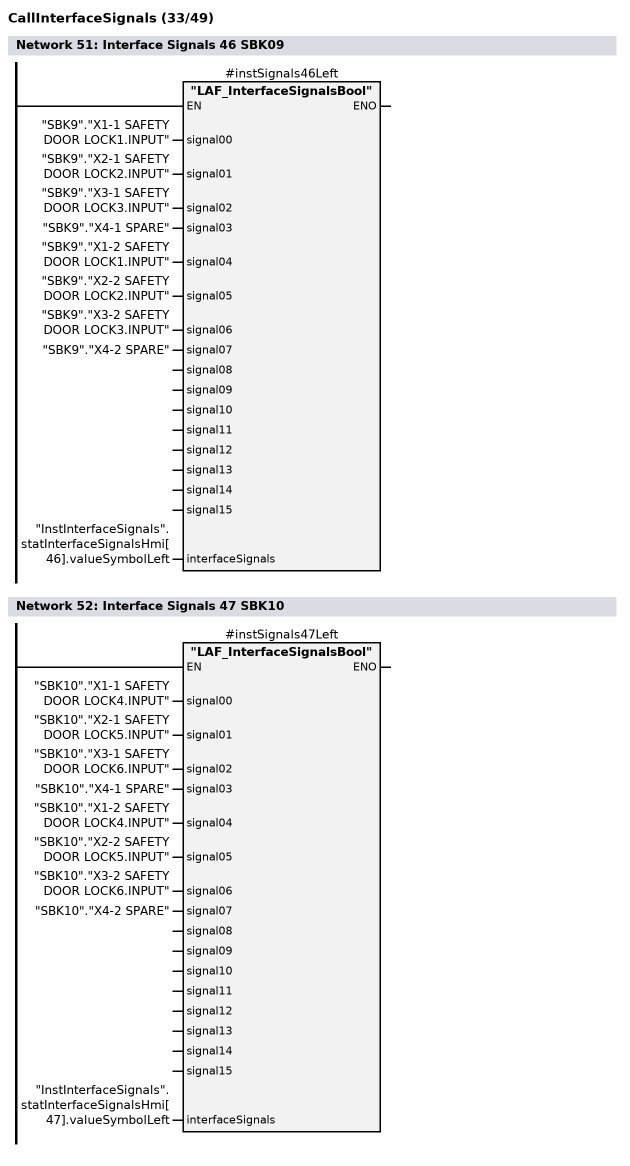
   RUNG wire#powerrail
      #instSignals46Left(signal00 := "SBK9"."X1-1 SAFETY DOOR LOCK1.INPUT", signal01 := "SBK9"."X2-1 SAFETY DOOR LOCK2.INPUT", signal02 := "SBK9"."X3-1 SAFETY DOOR LOCK3.INPUT", signal03 := "SBK9"."X4-1 SPARE", signal04 := "SBK9"."X1-2 SAFETY DOOR LOCK1.INPUT", signal05 := "SBK9"."X2-2 SAFETY DOOR LOCK2.INPUT", signal06 := "SBK9"."X3-2 SAFETY DOOR LOCK3.INPUT", signal07 := "SBK9"."X4-2 SPARE", signal08 :=, signal09 :=, signal10 :=, signal11 :=, signal12 :=, signal13 :=, signal14 :=, signal15 :=, interfaceSignals := "InstInterfaceSignals".statInterfaceSignalsHmi[46].valueSymbolLeft)
   END_RUNG
   // the same network as SCL:
   #instSignals46Left(signal00 := "SBK9"."X1-1 SAFETY DOOR LOCK1.INPUT",   // "LAF_InterfaceSignalsBool"
                      signal01 := "SBK9"."X2-1 SAFETY DOOR LOCK2.INPUT",
                      signal02 := "SBK9"."X3-1 SAFETY DOOR LOCK3.INPUT",
                      signal03 := "SBK9"."X4-1 SPARE",
                      signal04 := "SBK9"."X1-2 SAFETY DOOR LOCK1.INPUT",
                      signal05 := "SBK9"."X2-2 SAFETY DOOR LOCK2.INPUT",
                      signal06 := "SBK9"."X3-2 SAFETY DOOR LOCK3.INPUT",
                      signal07 := "SBK9"."X4-2 SPARE",
                      interfaceSignals := "InstInterfaceSignals".statInterfaceSignalsHmi[46].valueSymbolLeft);
END_REGION

REGION Network 52: Interface Signals 47 SBK10
   RUNG wire#powerrail
      #instSignals47Left(signal00 := "SBK10"."X1-1 SAFETY DOOR LOCK4.INPUT", signal01 := "SBK10"."X2-1 SAFETY DOOR LOCK5.INPUT", signal02 := "SBK10"."X3-1 SAFETY DOOR LOCK6.INPUT", signal03 := "SBK10"."X4-1 SPARE", signal04 := "SBK10"."X1-2 SAFETY DOOR LOCK4.INPUT", signal05 := "SBK10"."X2-2 SAFETY DOOR LOCK5.INPUT", signal06 := "SBK10"."X3-2 SAFETY DOOR LOCK6.INPUT", signal07 := "SBK10"."X4-2 SPARE", signal08 :=, signal09 :=, signal10 :=, signal11 :=, signal12 :=, signal13 :=, signal14 :=, signal15 :=, interfaceSignals := "InstInterfaceSignals".statInterfaceSignalsHmi[47].valueSymbolLeft)
   END_RUNG
   // the same network as SCL:
   #instSignals47Left(signal00 := "SBK10"."X1-1 SAFETY DOOR LOCK4.INPUT",   // "LAF_InterfaceSignalsBool"
                      signal01 := "SBK10"."X2-1 SAFETY DOOR LOCK5.INPUT",
                      signal02 := "SBK10"."X3-1 SAFETY DOOR LOCK6.INPUT",
                      signal03 := "SBK10"."X4-1 SPARE",
                      signal04 := "SBK10"."X1-2 SAFETY DOOR LOCK4.INPUT",
                      signal05 := "SBK10"."X2-2 SAFETY DOOR LOCK5.INPUT",
                      signal06 := "SBK10"."X3-2 SAFETY DOOR LOCK6.INPUT",
                      signal07 := "SBK10"."X4-2 SPARE",
                      interfaceSignals := "InstInterfaceSignals".statInterfaceSignalsHmi[47].valueSymbolLeft);
END_REGION

REGION Network 53: Interface Signals 48 SBK11
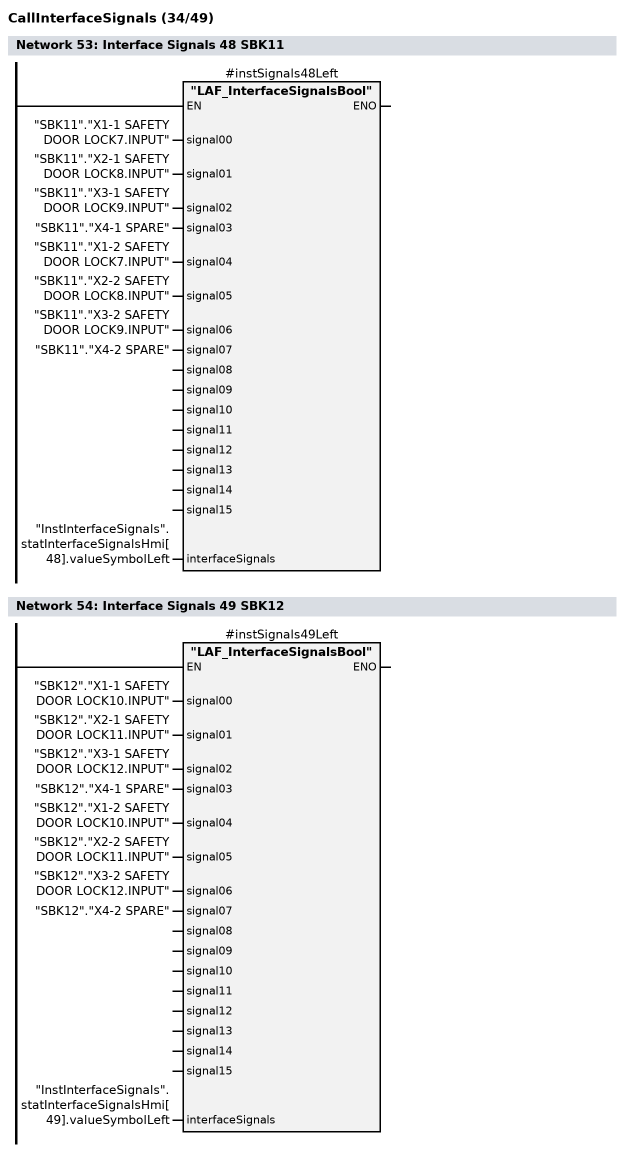
   RUNG wire#powerrail
      #instSignals48Left(signal00 := "SBK11"."X1-1 SAFETY DOOR LOCK7.INPUT", signal01 := "SBK11"."X2-1 SAFETY DOOR LOCK8.INPUT", signal02 := "SBK11"."X3-1 SAFETY DOOR LOCK9.INPUT", signal03 := "SBK11"."X4-1 SPARE", signal04 := "SBK11"."X1-2 SAFETY DOOR LOCK7.INPUT", signal05 := "SBK11"."X2-2 SAFETY DOOR LOCK8.INPUT", signal06 := "SBK11"."X3-2 SAFETY DOOR LOCK9.INPUT", signal07 := "SBK11"."X4-2 SPARE", signal08 :=, signal09 :=, signal10 :=, signal11 :=, signal12 :=, signal13 :=, signal14 :=, signal15 :=, interfaceSignals := "InstInterfaceSignals".statInterfaceSignalsHmi[48].valueSymbolLeft)
   END_RUNG
   // the same network as SCL:
   #instSignals48Left(signal00 := "SBK11"."X1-1 SAFETY DOOR LOCK7.INPUT",   // "LAF_InterfaceSignalsBool"
                      signal01 := "SBK11"."X2-1 SAFETY DOOR LOCK8.INPUT",
                      signal02 := "SBK11"."X3-1 SAFETY DOOR LOCK9.INPUT",
                      signal03 := "SBK11"."X4-1 SPARE",
                      signal04 := "SBK11"."X1-2 SAFETY DOOR LOCK7.INPUT",
                      signal05 := "SBK11"."X2-2 SAFETY DOOR LOCK8.INPUT",
                      signal06 := "SBK11"."X3-2 SAFETY DOOR LOCK9.INPUT",
                      signal07 := "SBK11"."X4-2 SPARE",
                      interfaceSignals := "InstInterfaceSignals".statInterfaceSignalsHmi[48].valueSymbolLeft);
END_REGION

REGION Network 54: Interface Signals 49 SBK12
   RUNG wire#powerrail
      #instSignals49Left(signal00 := "SBK12"."X1-1 SAFETY DOOR LOCK10.INPUT", signal01 := "SBK12"."X2-1 SAFETY DOOR LOCK11.INPUT", signal02 := "SBK12"."X3-1 SAFETY DOOR LOCK12.INPUT", signal03 := "SBK12"."X4-1 SPARE", signal04 := "SBK12"."X1-2 SAFETY DOOR LOCK10.INPUT", signal05 := "SBK12"."X2-2 SAFETY DOOR LOCK11.INPUT", signal06 := "SBK12"."X3-2 SAFETY DOOR LOCK12.INPUT", signal07 := "SBK12"."X4-2 SPARE", signal08 :=, signal09 :=, signal10 :=, signal11 :=, signal12 :=, signal13 :=, signal14 :=, signal15 :=, interfaceSignals := "InstInterfaceSignals".statInterfaceSignalsHmi[49].valueSymbolLeft)
   END_RUNG
   // the same network as SCL:
   #instSignals49Left(signal00 := "SBK12"."X1-1 SAFETY DOOR LOCK10.INPUT",   // "LAF_InterfaceSignalsBool"
                      signal01 := "SBK12"."X2-1 SAFETY DOOR LOCK11.INPUT",
                      signal02 := "SBK12"."X3-1 SAFETY DOOR LOCK12.INPUT",
                      signal03 := "SBK12"."X4-1 SPARE",
                      signal04 := "SBK12"."X1-2 SAFETY DOOR LOCK10.INPUT",
                      signal05 := "SBK12"."X2-2 SAFETY DOOR LOCK11.INPUT",
                      signal06 := "SBK12"."X3-2 SAFETY DOOR LOCK12.INPUT",
                      signal07 := "SBK12"."X4-2 SPARE",
                      interfaceSignals := "InstInterfaceSignals".statInterfaceSignalsHmi[49].valueSymbolLeft);
END_REGION

REGION Network 55: Interface Signals 50 SBK13
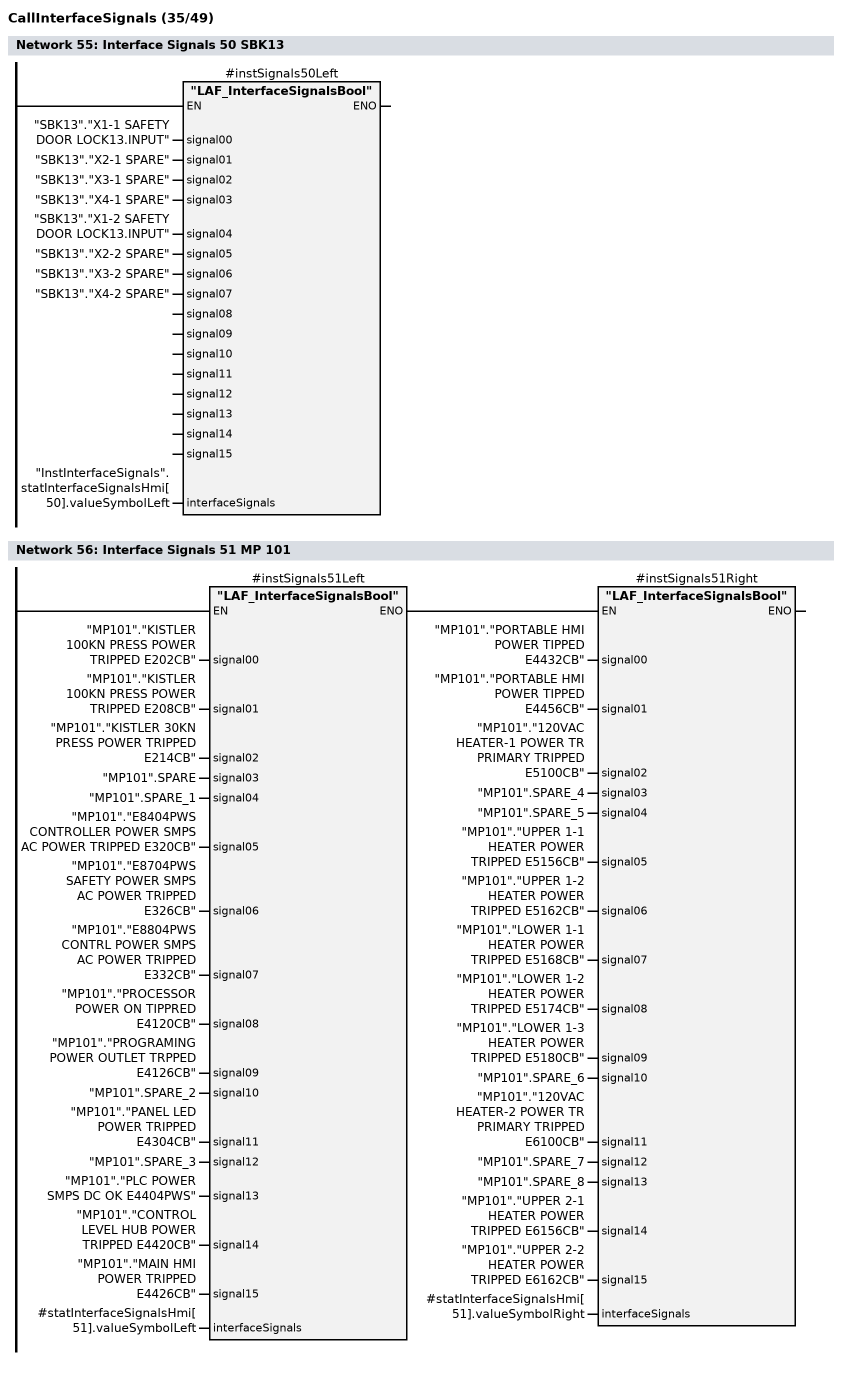
   RUNG wire#powerrail
      #instSignals50Left(signal00 := "SBK13"."X1-1 SAFETY DOOR LOCK13.INPUT", signal01 := "SBK13"."X2-1 SPARE", signal02 := "SBK13"."X3-1 SPARE", signal03 := "SBK13"."X4-1 SPARE", signal04 := "SBK13"."X1-2 SAFETY DOOR LOCK13.INPUT", signal05 := "SBK13"."X2-2 SPARE", signal06 := "SBK13"."X3-2 SPARE", signal07 := "SBK13"."X4-2 SPARE", signal08 :=, signal09 :=, signal10 :=, signal11 :=, signal12 :=, signal13 :=, signal14 :=, signal15 :=, interfaceSignals := "InstInterfaceSignals".statInterfaceSignalsHmi[50].valueSymbolLeft)
   END_RUNG
   // the same network as SCL:
   #instSignals50Left(signal00 := "SBK13"."X1-1 SAFETY DOOR LOCK13.INPUT",   // "LAF_InterfaceSignalsBool"
                      signal01 := "SBK13"."X2-1 SPARE",
                      signal02 := "SBK13"."X3-1 SPARE",
                      signal03 := "SBK13"."X4-1 SPARE",
                      signal04 := "SBK13"."X1-2 SAFETY DOOR LOCK13.INPUT",
                      signal05 := "SBK13"."X2-2 SPARE",
                      signal06 := "SBK13"."X3-2 SPARE",
                      signal07 := "SBK13"."X4-2 SPARE",
                      interfaceSignals := "InstInterfaceSignals".statInterfaceSignalsHmi[50].valueSymbolLeft);
END_REGION

REGION Network 56: Interface Signals 51 MP 101
   RUNG wire#powerrail
      #instSignals51Left(signal00 := "MP101"."KISTLER 100KN PRESS POWER TRIPPED E202CB", signal01 := "MP101"."KISTLER 100KN PRESS POWER TRIPPED E208CB", signal02 := "MP101"."KISTLER 30KN PRESS POWER TRIPPED E214CB", signal03 := "MP101".SPARE, signal04 := "MP101".SPARE_1, signal05 := "MP101"."E8404PWS CONTROLLER POWER SMPS AC POWER TRIPPED E320CB", signal06 := "MP101"."E8704PWS SAFETY POWER SMPS AC POWER TRIPPED E326CB", signal07 := "MP101"."E8804PWS CONTRL POWER SMPS AC POWER TRIPPED E332CB", signal08 := "MP101"."PROCESSOR POWER ON TIPPRED E4120CB", signal09 := "MP101"."PROGRAMING POWER OUTLET TRPPED E4126CB", signal10 := "MP101".SPARE_2, signal11 := "MP101"."PANEL LED POWER TRIPPED E4304CB", signal12 := "MP101".SPARE_3, signal13 := "MP101"."PLC POWER SMPS DC OK E4404PWS", signal14 := "MP101"."CONTROL LEVEL HUB POWER TRIPPED E4420CB", signal15 := "MP101"."MAIN HMI POWER TRIPPED E4426CB", interfaceSignals := #statInterfaceSignalsHmi[51].valueSymbolLeft)
      #instSignals51Right(signal00 := "MP101"."PORTABLE HMI POWER TIPPED E4432CB", signal01 := "MP101"."PORTABLE HMI POWER TIPPED E4456CB", signal02 := "MP101"."120VAC HEATER-1 POWER TR PRIMARY TRIPPED E5100CB", signal03 := "MP101".SPARE_4, signal04 := "MP101".SPARE_5, signal05 := "MP101"."UPPER 1-1 HEATER POWER TRIPPED E5156CB", signal06 := "MP101"."UPPER 1-2 HEATER POWER TRIPPED E5162CB", signal07 := "MP101"."LOWER 1-1 HEATER POWER TRIPPED E5168CB", signal08 := "MP101"."LOWER 1-2 HEATER POWER TRIPPED E5174CB", signal09 := "MP101"."LOWER 1-3 HEATER POWER TRIPPED E5180CB", signal10 := "MP101".SPARE_6, signal11 := "MP101"."120VAC HEATER-2 POWER TR PRIMARY TRIPPED E6100CB", signal12 := "MP101".SPARE_7, signal13 := "MP101".SPARE_8, signal14 := "MP101"."UPPER 2-1 HEATER POWER TRIPPED E6156CB", signal15 := "MP101"."UPPER 2-2 HEATER POWER TRIPPED E6162CB", interfaceSignals := #statInterfaceSignalsHmi[51].valueSymbolRight)
   END_RUNG
   // the same network as SCL:
   #instSignals51Left(signal00 := "MP101"."KISTLER 100KN PRESS POWER TRIPPED E202CB",   // "LAF_InterfaceSignalsBool"
                      signal01 := "MP101"."KISTLER 100KN PRESS POWER TRIPPED E208CB",
                      signal02 := "MP101"."KISTLER 30KN PRESS POWER TRIPPED E214CB",
                      signal03 := "MP101".SPARE,
                      signal04 := "MP101".SPARE_1,
                      signal05 := "MP101"."E8404PWS CONTROLLER POWER SMPS AC POWER TRIPPED E320CB",
                      signal06 := "MP101"."E8704PWS SAFETY POWER SMPS AC POWER TRIPPED E326CB",
                      signal07 := "MP101"."E8804PWS CONTRL POWER SMPS AC POWER TRIPPED E332CB",
                      signal08 := "MP101"."PROCESSOR POWER ON TIPPRED E4120CB",
                      signal09 := "MP101"."PROGRAMING POWER OUTLET TRPPED E4126CB",
                      signal10 := "MP101".SPARE_2,
                      signal11 := "MP101"."PANEL LED POWER TRIPPED E4304CB",
                      signal12 := "MP101".SPARE_3,
                      signal13 := "MP101"."PLC POWER SMPS DC OK E4404PWS",
                      signal14 := "MP101"."CONTROL LEVEL HUB POWER TRIPPED E4420CB",
                      signal15 := "MP101"."MAIN HMI POWER TRIPPED E4426CB",
                      interfaceSignals := #statInterfaceSignalsHmi[51].valueSymbolLeft,
                      ENO => #_w1);
   IF #_w1 THEN
       #instSignals51Right(signal00 := "MP101"."PORTABLE HMI POWER TIPPED E4432CB",   // "LAF_InterfaceSignalsBool"
                           signal01 := "MP101"."PORTABLE HMI POWER TIPPED E4456CB",
                           signal02 := "MP101"."120VAC HEATER-1 POWER TR PRIMARY TRIPPED E5100CB",
                           signal03 := "MP101".SPARE_4,
                           signal04 := "MP101".SPARE_5,
                           signal05 := "MP101"."UPPER 1-1 HEATER POWER TRIPPED E5156CB",
                           signal06 := "MP101"."UPPER 1-2 HEATER POWER TRIPPED E5162CB",
                           signal07 := "MP101"."LOWER 1-1 HEATER POWER TRIPPED E5168CB",
                           signal08 := "MP101"."LOWER 1-2 HEATER POWER TRIPPED E5174CB",
                           signal09 := "MP101"."LOWER 1-3 HEATER POWER TRIPPED E5180CB",
                           signal10 := "MP101".SPARE_6,
                           signal11 := "MP101"."120VAC HEATER-2 POWER TR PRIMARY TRIPPED E6100CB",
                           signal12 := "MP101".SPARE_7,
                           signal13 := "MP101".SPARE_8,
                           signal14 := "MP101"."UPPER 2-1 HEATER POWER TRIPPED E6156CB",
                           signal15 := "MP101"."UPPER 2-2 HEATER POWER TRIPPED E6162CB",
                           interfaceSignals := #statInterfaceSignalsHmi[51].valueSymbolRight);
   END_IF;
END_REGION

REGION Network 57: Interface Signals 52 MP 102
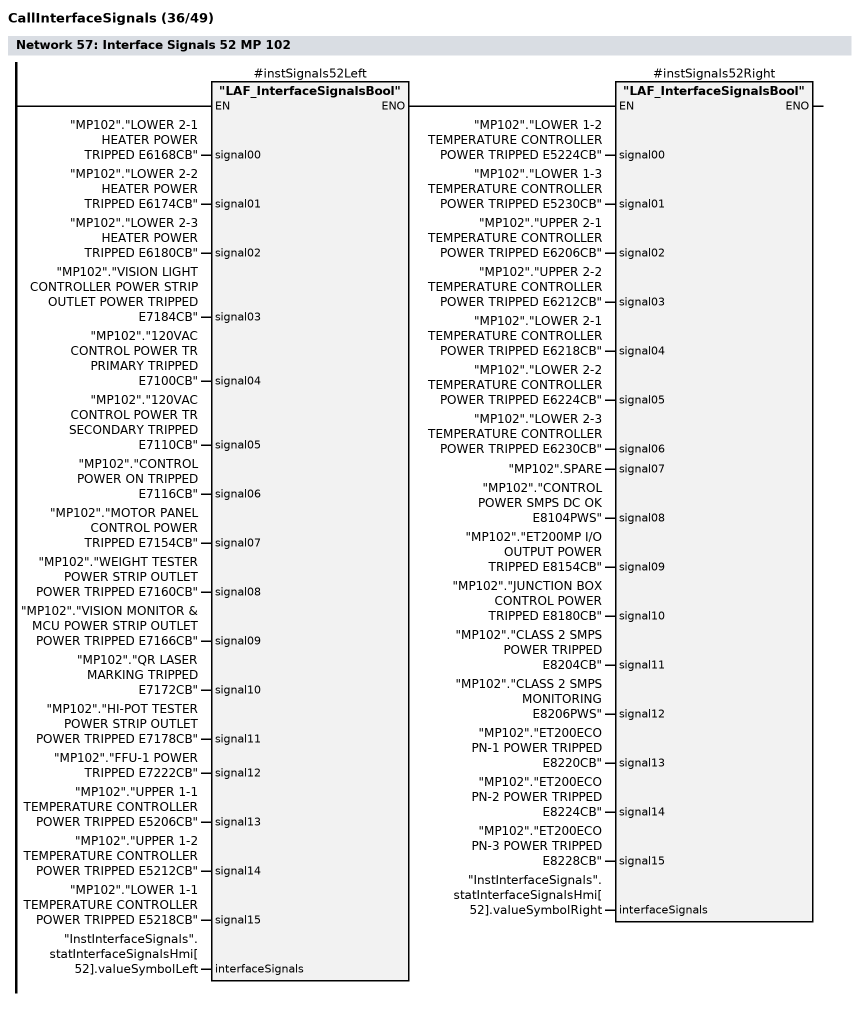
   RUNG wire#powerrail
      #instSignals52Left(signal00 := "MP102"."LOWER 2-1 HEATER POWER TRIPPED E6168CB", signal01 := "MP102"."LOWER 2-2 HEATER POWER TRIPPED E6174CB", signal02 := "MP102"."LOWER 2-3 HEATER POWER TRIPPED E6180CB", signal03 := "MP102"."VISION LIGHT CONTROLLER POWER STRIP OUTLET POWER TRIPPED E7184CB", signal04 := "MP102"."120VAC CONTROL POWER TR PRIMARY TRIPPED E7100CB", signal05 := "MP102"."120VAC CONTROL POWER TR SECONDARY TRIPPED E7110CB", signal06 := "MP102"."CONTROL POWER ON TRIPPED E7116CB", signal07 := "MP102"."MOTOR PANEL CONTROL POWER TRIPPED E7154CB", signal08 := "MP102"."WEIGHT TESTER POWER STRIP OUTLET POWER TRIPPED E7160CB", signal09 := "MP102"."VISION MONITOR & MCU POWER STRIP OUTLET POWER TRIPPED E7166CB", signal10 := "MP102"."QR LASER MARKING TRIPPED E7172CB", signal11 := "MP102"."HI-POT TESTER POWER STRIP OUTLET POWER TRIPPED E7178CB", signal12 := "MP102"."FFU-1 POWER TRIPPED E7222CB", signal13 := "MP102"."UPPER 1-1 TEMPERATURE CONTROLLER POWER TRIPPED E5206CB", signal14 := "MP102"."UPPER 1-2 TEMPERATURE CONTROLLER POWER TRIPPED E5212CB", signal15 := "MP102"."LOWER 1-1 TEMPERATURE CONTROLLER POWER TRIPPED E5218CB", interfaceSignals := "InstInterfaceSignals".statInterfaceSignalsHmi[52].valueSymbolLeft)
      #instSignals52Right(signal00 := "MP102"."LOWER 1-2 TEMPERATURE CONTROLLER POWER TRIPPED E5224CB", signal01 := "MP102"."LOWER 1-3 TEMPERATURE CONTROLLER POWER TRIPPED E5230CB", signal02 := "MP102"."UPPER 2-1 TEMPERATURE CONTROLLER POWER TRIPPED E6206CB", signal03 := "MP102"."UPPER 2-2 TEMPERATURE CONTROLLER POWER TRIPPED E6212CB", signal04 := "MP102"."LOWER 2-1 TEMPERATURE CONTROLLER POWER TRIPPED E6218CB", signal05 := "MP102"."LOWER 2-2 TEMPERATURE CONTROLLER POWER TRIPPED E6224CB", signal06 := "MP102"."LOWER 2-3 TEMPERATURE CONTROLLER POWER TRIPPED E6230CB", signal07 := "MP102".SPARE, signal08 := "MP102"."CONTROL POWER SMPS DC OK E8104PWS", signal09 := "MP102"."ET200MP I/O OUTPUT POWER TRIPPED E8154CB", signal10 := "MP102"."JUNCTION BOX CONTROL POWER TRIPPED E8180CB", signal11 := "MP102"."CLASS 2 SMPS POWER TRIPPED E8204CB", signal12 := "MP102"."CLASS 2 SMPS MONITORING E8206PWS", signal13 := "MP102"."ET200ECO PN-1 POWER TRIPPED E8220CB", signal14 := "MP102"."ET200ECO PN-2 POWER TRIPPED E8224CB", signal15 := "MP102"."ET200ECO PN-3 POWER TRIPPED E8228CB", interfaceSignals := "InstInterfaceSignals".statInterfaceSignalsHmi[52].valueSymbolRight)
   END_RUNG
   // the same network as SCL:
   #instSignals52Left(signal00 := "MP102"."LOWER 2-1 HEATER POWER TRIPPED E6168CB",   // "LAF_InterfaceSignalsBool"
                      signal01 := "MP102"."LOWER 2-2 HEATER POWER TRIPPED E6174CB",
                      signal02 := "MP102"."LOWER 2-3 HEATER POWER TRIPPED E6180CB",
                      signal03 := "MP102"."VISION LIGHT CONTROLLER POWER STRIP OUTLET POWER TRIPPED E7184CB",
                      signal04 := "MP102"."120VAC CONTROL POWER TR PRIMARY TRIPPED E7100CB",
                      signal05 := "MP102"."120VAC CONTROL POWER TR SECONDARY TRIPPED E7110CB",
                      signal06 := "MP102"."CONTROL POWER ON TRIPPED E7116CB",
                      signal07 := "MP102"."MOTOR PANEL CONTROL POWER TRIPPED E7154CB",
                      signal08 := "MP102"."WEIGHT TESTER POWER STRIP OUTLET POWER TRIPPED E7160CB",
                      signal09 := "MP102"."VISION MONITOR & MCU POWER STRIP OUTLET POWER TRIPPED E7166CB",
                      signal10 := "MP102"."QR LASER MARKING TRIPPED E7172CB",
                      signal11 := "MP102"."HI-POT TESTER POWER STRIP OUTLET POWER TRIPPED E7178CB",
                      signal12 := "MP102"."FFU-1 POWER TRIPPED E7222CB",
                      signal13 := "MP102"."UPPER 1-1 TEMPERATURE CONTROLLER POWER TRIPPED E5206CB",
                      signal14 := "MP102"."UPPER 1-2 TEMPERATURE CONTROLLER POWER TRIPPED E5212CB",
                      signal15 := "MP102"."LOWER 1-1 TEMPERATURE CONTROLLER POWER TRIPPED E5218CB",
                      interfaceSignals := "InstInterfaceSignals".statInterfaceSignalsHmi[52].valueSymbolLeft,
                      ENO => #_w1);
   IF #_w1 THEN
       #instSignals52Right(signal00 := "MP102"."LOWER 1-2 TEMPERATURE CONTROLLER POWER TRIPPED E5224CB",   // "LAF_InterfaceSignalsBool"
                           signal01 := "MP102"."LOWER 1-3 TEMPERATURE CONTROLLER POWER TRIPPED E5230CB",
                           signal02 := "MP102"."UPPER 2-1 TEMPERATURE CONTROLLER POWER TRIPPED E6206CB",
                           signal03 := "MP102"."UPPER 2-2 TEMPERATURE CONTROLLER POWER TRIPPED E6212CB",
                           signal04 := "MP102"."LOWER 2-1 TEMPERATURE CONTROLLER POWER TRIPPED E6218CB",
                           signal05 := "MP102"."LOWER 2-2 TEMPERATURE CONTROLLER POWER TRIPPED E6224CB",
                           signal06 := "MP102"."LOWER 2-3 TEMPERATURE CONTROLLER POWER TRIPPED E6230CB",
                           signal07 := "MP102".SPARE,
                           signal08 := "MP102"."CONTROL POWER SMPS DC OK E8104PWS",
                           signal09 := "MP102"."ET200MP I/O OUTPUT POWER TRIPPED E8154CB",
                           signal10 := "MP102"."JUNCTION BOX CONTROL POWER TRIPPED E8180CB",
                           signal11 := "MP102"."CLASS 2 SMPS POWER TRIPPED E8204CB",
                           signal12 := "MP102"."CLASS 2 SMPS MONITORING E8206PWS",
                           signal13 := "MP102"."ET200ECO PN-1 POWER TRIPPED E8220CB",
                           signal14 := "MP102"."ET200ECO PN-2 POWER TRIPPED E8224CB",
                           signal15 := "MP102"."ET200ECO PN-3 POWER TRIPPED E8228CB",
                           interfaceSignals := "InstInterfaceSignals".statInterfaceSignalsHmi[52].valueSymbolRight);
   END_IF;
END_REGION

REGION Network 58: Interface Signals 53 MP 103
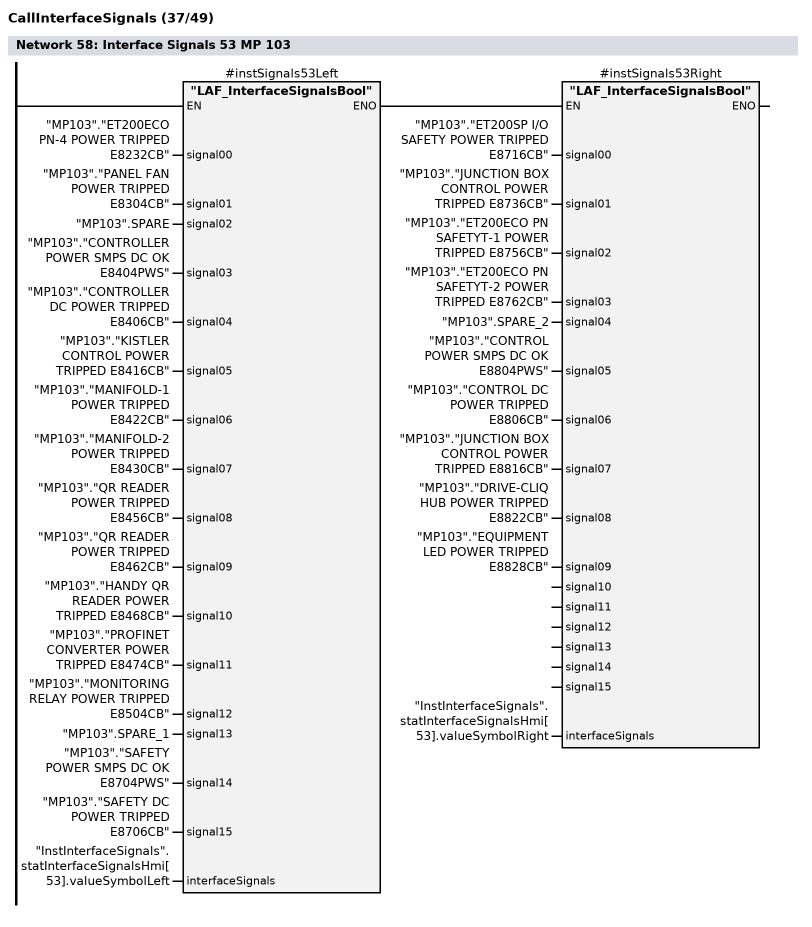
   RUNG wire#powerrail
      #instSignals53Left(signal00 := "MP103"."ET200ECO PN-4 POWER TRIPPED E8232CB", signal01 := "MP103"."PANEL FAN POWER TRIPPED E8304CB", signal02 := "MP103".SPARE, signal03 := "MP103"."CONTROLLER POWER SMPS DC OK E8404PWS", signal04 := "MP103"."CONTROLLER DC POWER TRIPPED E8406CB", signal05 := "MP103"."KISTLER CONTROL POWER TRIPPED E8416CB", signal06 := "MP103"."MANIFOLD-1 POWER TRIPPED E8422CB", signal07 := "MP103"."MANIFOLD-2 POWER TRIPPED E8430CB", signal08 := "MP103"."QR READER POWER TRIPPED E8456CB", signal09 := "MP103"."QR READER POWER TRIPPED E8462CB", signal10 := "MP103"."HANDY QR READER POWER TRIPPED E8468CB", signal11 := "MP103"."PROFINET CONVERTER POWER TRIPPED E8474CB", signal12 := "MP103"."MONITORING RELAY POWER TRIPPED E8504CB", signal13 := "MP103".SPARE_1, signal14 := "MP103"."SAFETY POWER SMPS DC OK E8704PWS", signal15 := "MP103"."SAFETY DC POWER TRIPPED E8706CB", interfaceSignals := "InstInterfaceSignals".statInterfaceSignalsHmi[53].valueSymbolLeft)
      #instSignals53Right(signal00 := "MP103"."ET200SP I/O SAFETY POWER TRIPPED E8716CB", signal01 := "MP103"."JUNCTION BOX CONTROL POWER TRIPPED E8736CB", signal02 := "MP103"."ET200ECO PN SAFETYT-1 POWER TRIPPED E8756CB", signal03 := "MP103"."ET200ECO PN SAFETYT-2 POWER TRIPPED E8762CB", signal04 := "MP103".SPARE_2, signal05 := "MP103"."CONTROL POWER SMPS DC OK E8804PWS", signal06 := "MP103"."CONTROL DC POWER TRIPPED E8806CB", signal07 := "MP103"."JUNCTION BOX CONTROL POWER TRIPPED E8816CB", signal08 := "MP103"."DRIVE-CLIQ HUB POWER TRIPPED E8822CB", signal09 := "MP103"."EQUIPMENT LED POWER TRIPPED E8828CB", signal10 :=, signal11 :=, signal12 :=, signal13 :=, signal14 :=, signal15 :=, interfaceSignals := "InstInterfaceSignals".statInterfaceSignalsHmi[53].valueSymbolRight)
   END_RUNG
   // the same network as SCL:
   #instSignals53Left(signal00 := "MP103"."ET200ECO PN-4 POWER TRIPPED E8232CB",   // "LAF_InterfaceSignalsBool"
                      signal01 := "MP103"."PANEL FAN POWER TRIPPED E8304CB",
                      signal02 := "MP103".SPARE,
                      signal03 := "MP103"."CONTROLLER POWER SMPS DC OK E8404PWS",
                      signal04 := "MP103"."CONTROLLER DC POWER TRIPPED E8406CB",
                      signal05 := "MP103"."KISTLER CONTROL POWER TRIPPED E8416CB",
                      signal06 := "MP103"."MANIFOLD-1 POWER TRIPPED E8422CB",
                      signal07 := "MP103"."MANIFOLD-2 POWER TRIPPED E8430CB",
                      signal08 := "MP103"."QR READER POWER TRIPPED E8456CB",
                      signal09 := "MP103"."QR READER POWER TRIPPED E8462CB",
                      signal10 := "MP103"."HANDY QR READER POWER TRIPPED E8468CB",
                      signal11 := "MP103"."PROFINET CONVERTER POWER TRIPPED E8474CB",
                      signal12 := "MP103"."MONITORING RELAY POWER TRIPPED E8504CB",
                      signal13 := "MP103".SPARE_1,
                      signal14 := "MP103"."SAFETY POWER SMPS DC OK E8704PWS",
                      signal15 := "MP103"."SAFETY DC POWER TRIPPED E8706CB",
                      interfaceSignals := "InstInterfaceSignals".statInterfaceSignalsHmi[53].valueSymbolLeft,
                      ENO => #_w1);
   IF #_w1 THEN
       #instSignals53Right(signal00 := "MP103"."ET200SP I/O SAFETY POWER TRIPPED E8716CB",   // "LAF_InterfaceSignalsBool"
                           signal01 := "MP103"."JUNCTION BOX CONTROL POWER TRIPPED E8736CB",
                           signal02 := "MP103"."ET200ECO PN SAFETYT-1 POWER TRIPPED E8756CB",
                           signal03 := "MP103"."ET200ECO PN SAFETYT-2 POWER TRIPPED E8762CB",
                           signal04 := "MP103".SPARE_2,
                           signal05 := "MP103"."CONTROL POWER SMPS DC OK E8804PWS",
                           signal06 := "MP103"."CONTROL DC POWER TRIPPED E8806CB",
                           signal07 := "MP103"."JUNCTION BOX CONTROL POWER TRIPPED E8816CB",
                           signal08 := "MP103"."DRIVE-CLIQ HUB POWER TRIPPED E8822CB",
                           signal09 := "MP103"."EQUIPMENT LED POWER TRIPPED E8828CB",
                           interfaceSignals := "InstInterfaceSignals".statInterfaceSignalsHmi[53].valueSymbolRight);
   END_IF;
END_REGION

REGION Network 59: Interface Signals 54 MP 104
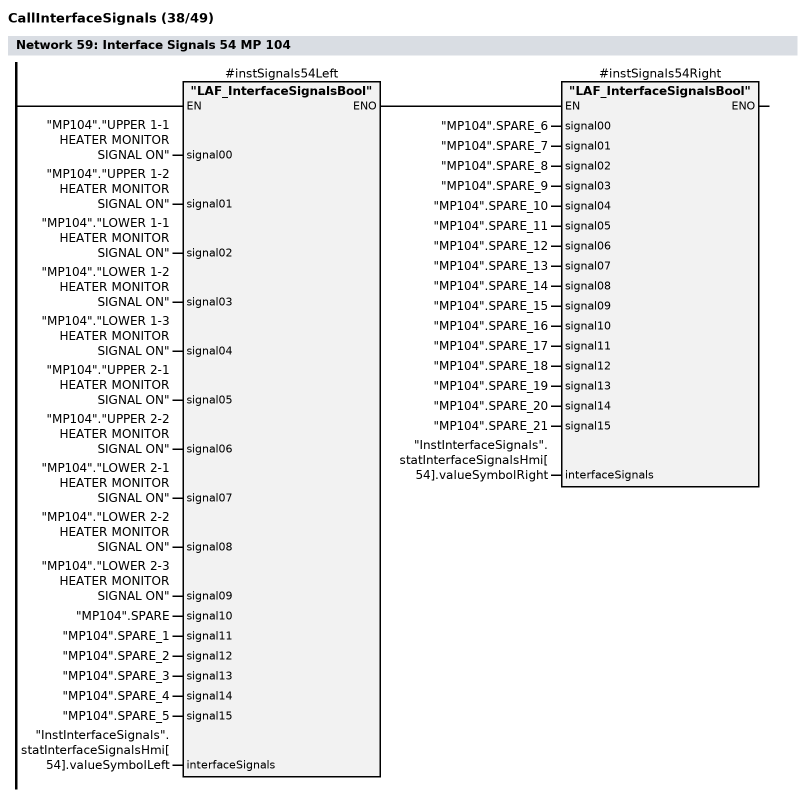
   RUNG wire#powerrail
      #instSignals54Left(signal00 := "MP104"."UPPER 1-1 HEATER MONITOR SIGNAL ON", signal01 := "MP104"."UPPER 1-2 HEATER MONITOR SIGNAL ON", signal02 := "MP104"."LOWER 1-1 HEATER MONITOR SIGNAL ON", signal03 := "MP104"."LOWER 1-2 HEATER MONITOR SIGNAL ON", signal04 := "MP104"."LOWER 1-3 HEATER MONITOR SIGNAL ON", signal05 := "MP104"."UPPER 2-1 HEATER MONITOR SIGNAL ON", signal06 := "MP104"."UPPER 2-2 HEATER MONITOR SIGNAL ON", signal07 := "MP104"."LOWER 2-1 HEATER MONITOR SIGNAL ON", signal08 := "MP104"."LOWER 2-2 HEATER MONITOR SIGNAL ON", signal09 := "MP104"."LOWER 2-3 HEATER MONITOR SIGNAL ON", signal10 := "MP104".SPARE, signal11 := "MP104".SPARE_1, signal12 := "MP104".SPARE_2, signal13 := "MP104".SPARE_3, signal14 := "MP104".SPARE_4, signal15 := "MP104".SPARE_5, interfaceSignals := "InstInterfaceSignals".statInterfaceSignalsHmi[54].valueSymbolLeft)
      #instSignals54Right(signal00 := "MP104".SPARE_6, signal01 := "MP104".SPARE_7, signal02 := "MP104".SPARE_8, signal03 := "MP104".SPARE_9, signal04 := "MP104".SPARE_10, signal05 := "MP104".SPARE_11, signal06 := "MP104".SPARE_12, signal07 := "MP104".SPARE_13, signal08 := "MP104".SPARE_14, signal09 := "MP104".SPARE_15, signal10 := "MP104".SPARE_16, signal11 := "MP104".SPARE_17, signal12 := "MP104".SPARE_18, signal13 := "MP104".SPARE_19, signal14 := "MP104".SPARE_20, signal15 := "MP104".SPARE_21, interfaceSignals := "InstInterfaceSignals".statInterfaceSignalsHmi[54].valueSymbolRight)
   END_RUNG
   // the same network as SCL:
   #instSignals54Left(signal00 := "MP104"."UPPER 1-1 HEATER MONITOR SIGNAL ON",   // "LAF_InterfaceSignalsBool"
                      signal01 := "MP104"."UPPER 1-2 HEATER MONITOR SIGNAL ON",
                      signal02 := "MP104"."LOWER 1-1 HEATER MONITOR SIGNAL ON",
                      signal03 := "MP104"."LOWER 1-2 HEATER MONITOR SIGNAL ON",
                      signal04 := "MP104"."LOWER 1-3 HEATER MONITOR SIGNAL ON",
                      signal05 := "MP104"."UPPER 2-1 HEATER MONITOR SIGNAL ON",
                      signal06 := "MP104"."UPPER 2-2 HEATER MONITOR SIGNAL ON",
                      signal07 := "MP104"."LOWER 2-1 HEATER MONITOR SIGNAL ON",
                      signal08 := "MP104"."LOWER 2-2 HEATER MONITOR SIGNAL ON",
                      signal09 := "MP104"."LOWER 2-3 HEATER MONITOR SIGNAL ON",
                      signal10 := "MP104".SPARE,
                      signal11 := "MP104".SPARE_1,
                      signal12 := "MP104".SPARE_2,
                      signal13 := "MP104".SPARE_3,
                      signal14 := "MP104".SPARE_4,
                      signal15 := "MP104".SPARE_5,
                      interfaceSignals := "InstInterfaceSignals".statInterfaceSignalsHmi[54].valueSymbolLeft,
                      ENO => #_w1);
   IF #_w1 THEN
       #instSignals54Right(signal00 := "MP104".SPARE_6,   // "LAF_InterfaceSignalsBool"
                           signal01 := "MP104".SPARE_7,
                           signal02 := "MP104".SPARE_8,
                           signal03 := "MP104".SPARE_9,
                           signal04 := "MP104".SPARE_10,
                           signal05 := "MP104".SPARE_11,
                           signal06 := "MP104".SPARE_12,
                           signal07 := "MP104".SPARE_13,
                           signal08 := "MP104".SPARE_14,
                           signal09 := "MP104".SPARE_15,
                           signal10 := "MP104".SPARE_16,
                           signal11 := "MP104".SPARE_17,
                           signal12 := "MP104".SPARE_18,
                           signal13 := "MP104".SPARE_19,
                           signal14 := "MP104".SPARE_20,
                           signal15 := "MP104".SPARE_21,
                           interfaceSignals := "InstInterfaceSignals".statInterfaceSignalsHmi[54].valueSymbolRight);
   END_IF;
END_REGION

REGION Network 60: Interface Signals 55 MP 105
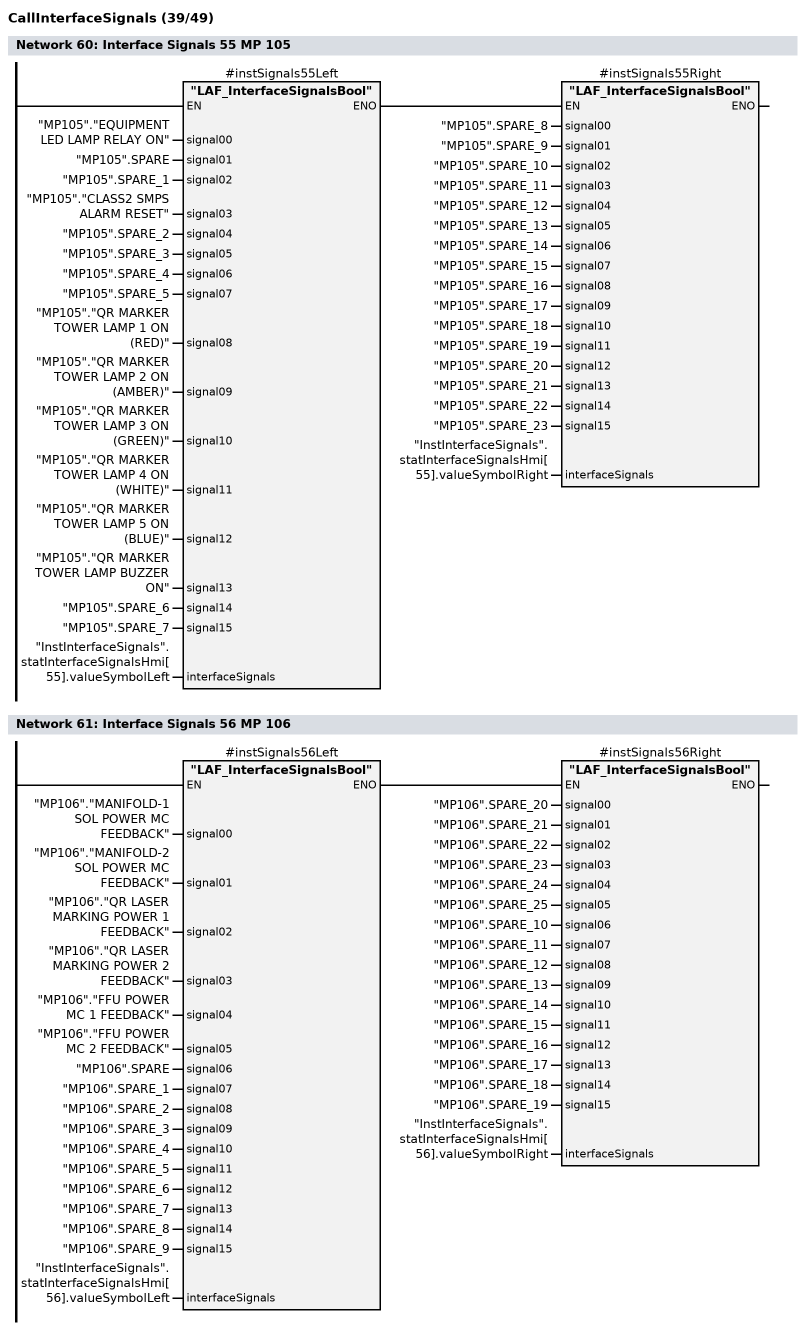
   RUNG wire#powerrail
      #instSignals55Left(signal00 := "MP105"."EQUIPMENT LED LAMP RELAY ON", signal01 := "MP105".SPARE, signal02 := "MP105".SPARE_1, signal03 := "MP105"."CLASS2 SMPS ALARM RESET", signal04 := "MP105".SPARE_2, signal05 := "MP105".SPARE_3, signal06 := "MP105".SPARE_4, signal07 := "MP105".SPARE_5, signal08 := "MP105"."QR MARKER TOWER LAMP 1 ON (RED)", signal09 := "MP105"."QR MARKER TOWER LAMP 2 ON (AMBER)", signal10 := "MP105"."QR MARKER TOWER LAMP 3 ON (GREEN)", signal11 := "MP105"."QR MARKER TOWER LAMP 4 ON (WHITE)", signal12 := "MP105"."QR MARKER TOWER LAMP 5 ON (BLUE)", signal13 := "MP105"."QR MARKER TOWER LAMP BUZZER ON", signal14 := "MP105".SPARE_6, signal15 := "MP105".SPARE_7, interfaceSignals := "InstInterfaceSignals".statInterfaceSignalsHmi[55].valueSymbolLeft)
      #instSignals55Right(signal00 := "MP105".SPARE_8, signal01 := "MP105".SPARE_9, signal02 := "MP105".SPARE_10, signal03 := "MP105".SPARE_11, signal04 := "MP105".SPARE_12, signal05 := "MP105".SPARE_13, signal06 := "MP105".SPARE_14, signal07 := "MP105".SPARE_15, signal08 := "MP105".SPARE_16, signal09 := "MP105".SPARE_17, signal10 := "MP105".SPARE_18, signal11 := "MP105".SPARE_19, signal12 := "MP105".SPARE_20, signal13 := "MP105".SPARE_21, signal14 := "MP105".SPARE_22, signal15 := "MP105".SPARE_23, interfaceSignals := "InstInterfaceSignals".statInterfaceSignalsHmi[55].valueSymbolRight)
   END_RUNG
   // the same network as SCL:
   #instSignals55Left(signal00 := "MP105"."EQUIPMENT LED LAMP RELAY ON",   // "LAF_InterfaceSignalsBool"
                      signal01 := "MP105".SPARE,
                      signal02 := "MP105".SPARE_1,
                      signal03 := "MP105"."CLASS2 SMPS ALARM RESET",
                      signal04 := "MP105".SPARE_2,
                      signal05 := "MP105".SPARE_3,
                      signal06 := "MP105".SPARE_4,
                      signal07 := "MP105".SPARE_5,
                      signal08 := "MP105"."QR MARKER TOWER LAMP 1 ON (RED)",
                      signal09 := "MP105"."QR MARKER TOWER LAMP 2 ON (AMBER)",
                      signal10 := "MP105"."QR MARKER TOWER LAMP 3 ON (GREEN)",
                      signal11 := "MP105"."QR MARKER TOWER LAMP 4 ON (WHITE)",
                      signal12 := "MP105"."QR MARKER TOWER LAMP 5 ON (BLUE)",
                      signal13 := "MP105"."QR MARKER TOWER LAMP BUZZER ON",
                      signal14 := "MP105".SPARE_6,
                      signal15 := "MP105".SPARE_7,
                      interfaceSignals := "InstInterfaceSignals".statInterfaceSignalsHmi[55].valueSymbolLeft,
                      ENO => #_w1);
   IF #_w1 THEN
       #instSignals55Right(signal00 := "MP105".SPARE_8,   // "LAF_InterfaceSignalsBool"
                           signal01 := "MP105".SPARE_9,
                           signal02 := "MP105".SPARE_10,
                           signal03 := "MP105".SPARE_11,
                           signal04 := "MP105".SPARE_12,
                           signal05 := "MP105".SPARE_13,
                           signal06 := "MP105".SPARE_14,
                           signal07 := "MP105".SPARE_15,
                           signal08 := "MP105".SPARE_16,
                           signal09 := "MP105".SPARE_17,
                           signal10 := "MP105".SPARE_18,
                           signal11 := "MP105".SPARE_19,
                           signal12 := "MP105".SPARE_20,
                           signal13 := "MP105".SPARE_21,
                           signal14 := "MP105".SPARE_22,
                           signal15 := "MP105".SPARE_23,
                           interfaceSignals := "InstInterfaceSignals".statInterfaceSignalsHmi[55].valueSymbolRight);
   END_IF;
END_REGION

REGION Network 61: Interface Signals 56 MP 106
   RUNG wire#powerrail
      #instSignals56Left(signal00 := "MP106"."MANIFOLD-1 SOL POWER MC FEEDBACK", signal01 := "MP106"."MANIFOLD-2 SOL POWER MC FEEDBACK", signal02 := "MP106"."QR LASER MARKING POWER 1 FEEDBACK", signal03 := "MP106"."QR LASER MARKING POWER 2 FEEDBACK", signal04 := "MP106"."FFU POWER MC 1 FEEDBACK", signal05 := "MP106"."FFU POWER MC 2 FEEDBACK", signal06 := "MP106".SPARE, signal07 := "MP106".SPARE_1, signal08 := "MP106".SPARE_2, signal09 := "MP106".SPARE_3, signal10 := "MP106".SPARE_4, signal11 := "MP106".SPARE_5, signal12 := "MP106".SPARE_6, signal13 := "MP106".SPARE_7, signal14 := "MP106".SPARE_8, signal15 := "MP106".SPARE_9, interfaceSignals := "InstInterfaceSignals".statInterfaceSignalsHmi[56].valueSymbolLeft)
      #instSignals56Right(signal00 := "MP106".SPARE_20, signal01 := "MP106".SPARE_21, signal02 := "MP106".SPARE_22, signal03 := "MP106".SPARE_23, signal04 := "MP106".SPARE_24, signal05 := "MP106".SPARE_25, signal06 := "MP106".SPARE_10, signal07 := "MP106".SPARE_11, signal08 := "MP106".SPARE_12, signal09 := "MP106".SPARE_13, signal10 := "MP106".SPARE_14, signal11 := "MP106".SPARE_15, signal12 := "MP106".SPARE_16, signal13 := "MP106".SPARE_17, signal14 := "MP106".SPARE_18, signal15 := "MP106".SPARE_19, interfaceSignals := "InstInterfaceSignals".statInterfaceSignalsHmi[56].valueSymbolRight)
   END_RUNG
   // the same network as SCL:
   #instSignals56Left(signal00 := "MP106"."MANIFOLD-1 SOL POWER MC FEEDBACK",   // "LAF_InterfaceSignalsBool"
                      signal01 := "MP106"."MANIFOLD-2 SOL POWER MC FEEDBACK",
                      signal02 := "MP106"."QR LASER MARKING POWER 1 FEEDBACK",
                      signal03 := "MP106"."QR LASER MARKING POWER 2 FEEDBACK",
                      signal04 := "MP106"."FFU POWER MC 1 FEEDBACK",
                      signal05 := "MP106"."FFU POWER MC 2 FEEDBACK",
                      signal06 := "MP106".SPARE,
                      signal07 := "MP106".SPARE_1,
                      signal08 := "MP106".SPARE_2,
                      signal09 := "MP106".SPARE_3,
                      signal10 := "MP106".SPARE_4,
                      signal11 := "MP106".SPARE_5,
                      signal12 := "MP106".SPARE_6,
                      signal13 := "MP106".SPARE_7,
                      signal14 := "MP106".SPARE_8,
                      signal15 := "MP106".SPARE_9,
                      interfaceSignals := "InstInterfaceSignals".statInterfaceSignalsHmi[56].valueSymbolLeft,
                      ENO => #_w1);
   IF #_w1 THEN
       #instSignals56Right(signal00 := "MP106".SPARE_20,   // "LAF_InterfaceSignalsBool"
                           signal01 := "MP106".SPARE_21,
                           signal02 := "MP106".SPARE_22,
                           signal03 := "MP106".SPARE_23,
                           signal04 := "MP106".SPARE_24,
                           signal05 := "MP106".SPARE_25,
                           signal06 := "MP106".SPARE_10,
                           signal07 := "MP106".SPARE_11,
                           signal08 := "MP106".SPARE_12,
                           signal09 := "MP106".SPARE_13,
                           signal10 := "MP106".SPARE_14,
                           signal11 := "MP106".SPARE_15,
                           signal12 := "MP106".SPARE_16,
                           signal13 := "MP106".SPARE_17,
                           signal14 := "MP106".SPARE_18,
                           signal15 := "MP106".SPARE_19,
                           interfaceSignals := "InstInterfaceSignals".statInterfaceSignalsHmi[56].valueSymbolRight);
   END_IF;
END_REGION

REGION Network 62: Interface Signals 57 MP 107
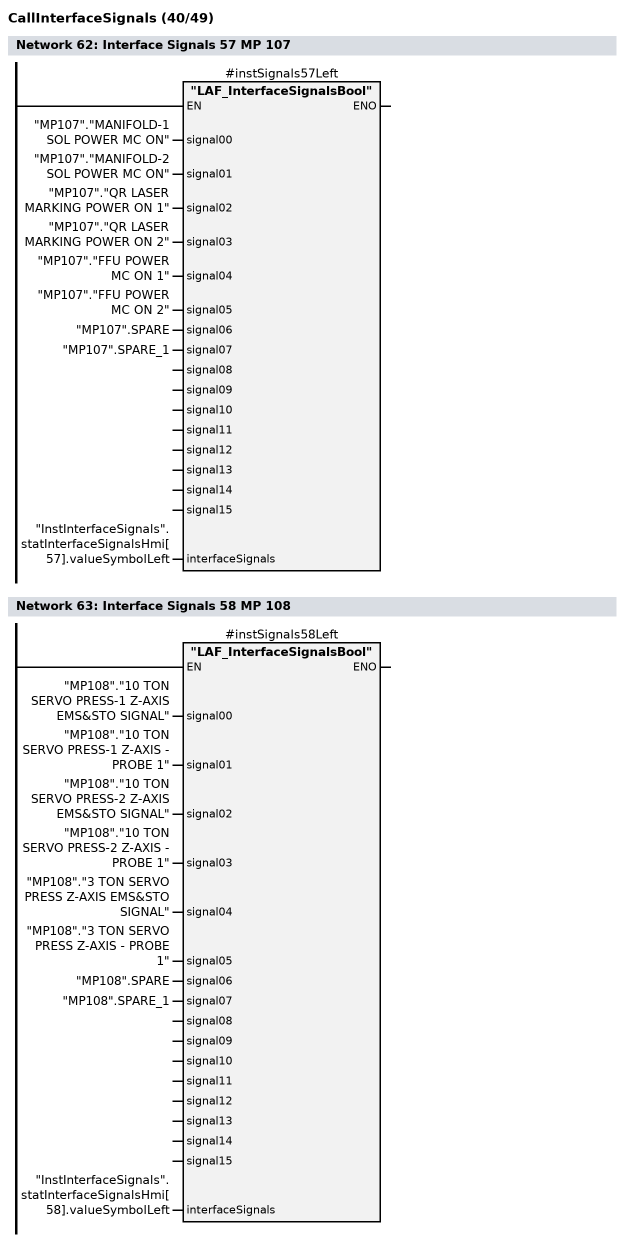
   RUNG wire#powerrail
      #instSignals57Left(signal00 := "MP107"."MANIFOLD-1 SOL POWER MC ON", signal01 := "MP107"."MANIFOLD-2 SOL POWER MC ON", signal02 := "MP107"."QR LASER MARKING POWER ON 1", signal03 := "MP107"."QR LASER MARKING POWER ON 2", signal04 := "MP107"."FFU POWER MC ON 1", signal05 := "MP107"."FFU POWER MC ON 2", signal06 := "MP107".SPARE, signal07 := "MP107".SPARE_1, signal08 :=, signal09 :=, signal10 :=, signal11 :=, signal12 :=, signal13 :=, signal14 :=, signal15 :=, interfaceSignals := "InstInterfaceSignals".statInterfaceSignalsHmi[57].valueSymbolLeft)
   END_RUNG
   // the same network as SCL:
   #instSignals57Left(signal00 := "MP107"."MANIFOLD-1 SOL POWER MC ON",   // "LAF_InterfaceSignalsBool"
                      signal01 := "MP107"."MANIFOLD-2 SOL POWER MC ON",
                      signal02 := "MP107"."QR LASER MARKING POWER ON 1",
                      signal03 := "MP107"."QR LASER MARKING POWER ON 2",
                      signal04 := "MP107"."FFU POWER MC ON 1",
                      signal05 := "MP107"."FFU POWER MC ON 2",
                      signal06 := "MP107".SPARE,
                      signal07 := "MP107".SPARE_1,
                      interfaceSignals := "InstInterfaceSignals".statInterfaceSignalsHmi[57].valueSymbolLeft);
END_REGION

REGION Network 63: Interface Signals 58 MP 108
   RUNG wire#powerrail
      #instSignals58Left(signal00 := "MP108"."10 TON SERVO PRESS-1 Z-AXIS EMS&STO SIGNAL", signal01 := "MP108"."10 TON SERVO PRESS-1 Z-AXIS - PROBE 1", signal02 := "MP108"."10 TON SERVO PRESS-2 Z-AXIS EMS&STO SIGNAL", signal03 := "MP108"."10 TON SERVO PRESS-2 Z-AXIS - PROBE 1", signal04 := "MP108"."3 TON SERVO PRESS Z-AXIS EMS&STO SIGNAL", signal05 := "MP108"."3 TON SERVO PRESS Z-AXIS - PROBE 1", signal06 := "MP108".SPARE, signal07 := "MP108".SPARE_1, signal08 :=, signal09 :=, signal10 :=, signal11 :=, signal12 :=, signal13 :=, signal14 :=, signal15 :=, interfaceSignals := "InstInterfaceSignals".statInterfaceSignalsHmi[58].valueSymbolLeft)
   END_RUNG
   // the same network as SCL:
   #instSignals58Left(signal00 := "MP108"."10 TON SERVO PRESS-1 Z-AXIS EMS&STO SIGNAL",   // "LAF_InterfaceSignalsBool"
                      signal01 := "MP108"."10 TON SERVO PRESS-1 Z-AXIS - PROBE 1",
                      signal02 := "MP108"."10 TON SERVO PRESS-2 Z-AXIS EMS&STO SIGNAL",
                      signal03 := "MP108"."10 TON SERVO PRESS-2 Z-AXIS - PROBE 1",
                      signal04 := "MP108"."3 TON SERVO PRESS Z-AXIS EMS&STO SIGNAL",
                      signal05 := "MP108"."3 TON SERVO PRESS Z-AXIS - PROBE 1",
                      signal06 := "MP108".SPARE,
                      signal07 := "MP108".SPARE_1,
                      interfaceSignals := "InstInterfaceSignals".statInterfaceSignalsHmi[58].valueSymbolLeft);
END_REGION

REGION Network 64: Interface Signals 59 MP 109
END_REGION

REGION Network 65: Interface Signals 60 SP 201
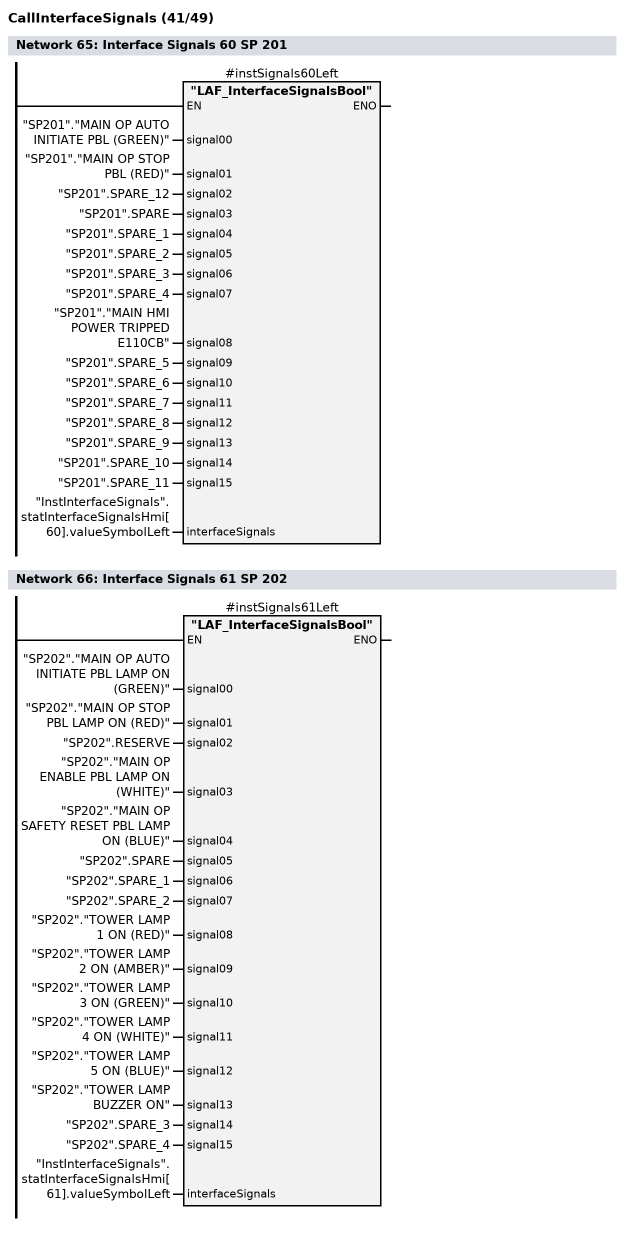
   RUNG wire#powerrail
      #instSignals60Left(signal00 := "SP201"."MAIN OP AUTO INITIATE PBL (GREEN)", signal01 := "SP201"."MAIN OP STOP PBL (RED)", signal02 := "SP201".SPARE_12, signal03 := "SP201".SPARE, signal04 := "SP201".SPARE_1, signal05 := "SP201".SPARE_2, signal06 := "SP201".SPARE_3, signal07 := "SP201".SPARE_4, signal08 := "SP201"."MAIN HMI POWER TRIPPED E110CB", signal09 := "SP201".SPARE_5, signal10 := "SP201".SPARE_6, signal11 := "SP201".SPARE_7, signal12 := "SP201".SPARE_8, signal13 := "SP201".SPARE_9, signal14 := "SP201".SPARE_10, signal15 := "SP201".SPARE_11, interfaceSignals := "InstInterfaceSignals".statInterfaceSignalsHmi[60].valueSymbolLeft)
   END_RUNG
   // the same network as SCL:
   #instSignals60Left(signal00 := "SP201"."MAIN OP AUTO INITIATE PBL (GREEN)",   // "LAF_InterfaceSignalsBool"
                      signal01 := "SP201"."MAIN OP STOP PBL (RED)",
                      signal02 := "SP201".SPARE_12,
                      signal03 := "SP201".SPARE,
                      signal04 := "SP201".SPARE_1,
                      signal05 := "SP201".SPARE_2,
                      signal06 := "SP201".SPARE_3,
                      signal07 := "SP201".SPARE_4,
                      signal08 := "SP201"."MAIN HMI POWER TRIPPED E110CB",
                      signal09 := "SP201".SPARE_5,
                      signal10 := "SP201".SPARE_6,
                      signal11 := "SP201".SPARE_7,
                      signal12 := "SP201".SPARE_8,
                      signal13 := "SP201".SPARE_9,
                      signal14 := "SP201".SPARE_10,
                      signal15 := "SP201".SPARE_11,
                      interfaceSignals := "InstInterfaceSignals".statInterfaceSignalsHmi[60].valueSymbolLeft);
END_REGION

REGION Network 66: Interface Signals 61 SP 202
   RUNG wire#powerrail
      #instSignals61Left(signal00 := "SP202"."MAIN OP AUTO INITIATE PBL LAMP ON (GREEN)", signal01 := "SP202"."MAIN OP STOP PBL LAMP ON (RED)", signal02 := "SP202".RESERVE, signal03 := "SP202"."MAIN OP ENABLE PBL LAMP ON (WHITE)", signal04 := "SP202"."MAIN OP SAFETY RESET PBL LAMP ON (BLUE)", signal05 := "SP202".SPARE, signal06 := "SP202".SPARE_1, signal07 := "SP202".SPARE_2, signal08 := "SP202"."TOWER LAMP 1 ON (RED)", signal09 := "SP202"."TOWER LAMP 2 ON (AMBER)", signal10 := "SP202"."TOWER LAMP 3 ON (GREEN)", signal11 := "SP202"."TOWER LAMP 4 ON (WHITE)", signal12 := "SP202"."TOWER LAMP 5 ON (BLUE)", signal13 := "SP202"."TOWER LAMP BUZZER ON", signal14 := "SP202".SPARE_3, signal15 := "SP202".SPARE_4, interfaceSignals := "InstInterfaceSignals".statInterfaceSignalsHmi[61].valueSymbolLeft)
   END_RUNG
   // the same network as SCL:
   #instSignals61Left(signal00 := "SP202"."MAIN OP AUTO INITIATE PBL LAMP ON (GREEN)",   // "LAF_InterfaceSignalsBool"
                      signal01 := "SP202"."MAIN OP STOP PBL LAMP ON (RED)",
                      signal02 := "SP202".RESERVE,
                      signal03 := "SP202"."MAIN OP ENABLE PBL LAMP ON (WHITE)",
                      signal04 := "SP202"."MAIN OP SAFETY RESET PBL LAMP ON (BLUE)",
                      signal05 := "SP202".SPARE,
                      signal06 := "SP202".SPARE_1,
                      signal07 := "SP202".SPARE_2,
                      signal08 := "SP202"."TOWER LAMP 1 ON (RED)",
                      signal09 := "SP202"."TOWER LAMP 2 ON (AMBER)",
                      signal10 := "SP202"."TOWER LAMP 3 ON (GREEN)",
                      signal11 := "SP202"."TOWER LAMP 4 ON (WHITE)",
                      signal12 := "SP202"."TOWER LAMP 5 ON (BLUE)",
                      signal13 := "SP202"."TOWER LAMP BUZZER ON",
                      signal14 := "SP202".SPARE_3,
                      signal15 := "SP202".SPARE_4,
                      interfaceSignals := "InstInterfaceSignals".statInterfaceSignalsHmi[61].valueSymbolLeft);
END_REGION

REGION Network 67: Interface Signals 62 SP 203
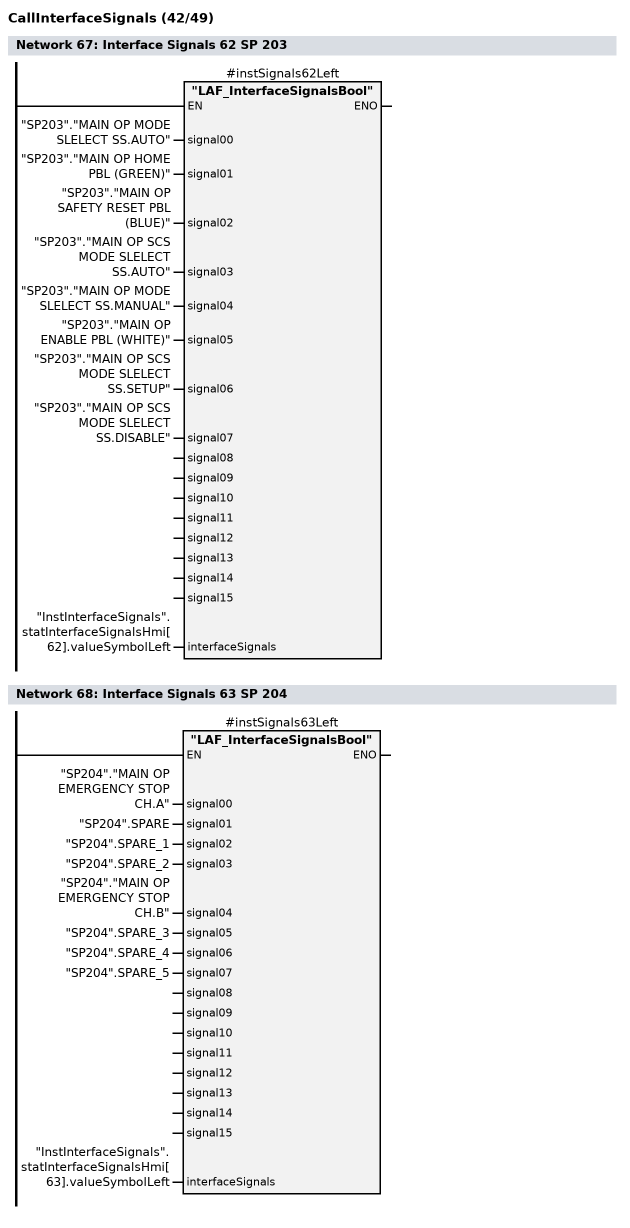
   RUNG wire#powerrail
      #instSignals62Left(signal00 := "SP203"."MAIN OP MODE SLELECT SS.AUTO", signal01 := "SP203"."MAIN OP HOME PBL (GREEN)", signal02 := "SP203"."MAIN OP SAFETY RESET PBL (BLUE)", signal03 := "SP203"."MAIN OP SCS MODE SLELECT SS.AUTO", signal04 := "SP203"."MAIN OP MODE SLELECT SS.MANUAL", signal05 := "SP203"."MAIN OP ENABLE PBL (WHITE)", signal06 := "SP203"."MAIN OP SCS MODE SLELECT SS.SETUP", signal07 := "SP203"."MAIN OP SCS MODE SLELECT SS.DISABLE", signal08 :=, signal09 :=, signal10 :=, signal11 :=, signal12 :=, signal13 :=, signal14 :=, signal15 :=, interfaceSignals := "InstInterfaceSignals".statInterfaceSignalsHmi[62].valueSymbolLeft)
   END_RUNG
   // the same network as SCL:
   #instSignals62Left(signal00 := "SP203"."MAIN OP MODE SLELECT SS.AUTO",   // "LAF_InterfaceSignalsBool"
                      signal01 := "SP203"."MAIN OP HOME PBL (GREEN)",
                      signal02 := "SP203"."MAIN OP SAFETY RESET PBL (BLUE)",
                      signal03 := "SP203"."MAIN OP SCS MODE SLELECT SS.AUTO",
                      signal04 := "SP203"."MAIN OP MODE SLELECT SS.MANUAL",
                      signal05 := "SP203"."MAIN OP ENABLE PBL (WHITE)",
                      signal06 := "SP203"."MAIN OP SCS MODE SLELECT SS.SETUP",
                      signal07 := "SP203"."MAIN OP SCS MODE SLELECT SS.DISABLE",
                      interfaceSignals := "InstInterfaceSignals".statInterfaceSignalsHmi[62].valueSymbolLeft);
END_REGION

REGION Network 68: Interface Signals 63 SP 204
   RUNG wire#powerrail
      #instSignals63Left(signal00 := "SP204"."MAIN OP EMERGENCY STOP CH.A", signal01 := "SP204".SPARE, signal02 := "SP204".SPARE_1, signal03 := "SP204".SPARE_2, signal04 := "SP204"."MAIN OP EMERGENCY STOP CH.B", signal05 := "SP204".SPARE_3, signal06 := "SP204".SPARE_4, signal07 := "SP204".SPARE_5, signal08 :=, signal09 :=, signal10 :=, signal11 :=, signal12 :=, signal13 :=, signal14 :=, signal15 :=, interfaceSignals := "InstInterfaceSignals".statInterfaceSignalsHmi[63].valueSymbolLeft)
   END_RUNG
   // the same network as SCL:
   #instSignals63Left(signal00 := "SP204"."MAIN OP EMERGENCY STOP CH.A",   // "LAF_InterfaceSignalsBool"
                      signal01 := "SP204".SPARE,
                      signal02 := "SP204".SPARE_1,
                      signal03 := "SP204".SPARE_2,
                      signal04 := "SP204"."MAIN OP EMERGENCY STOP CH.B",
                      signal05 := "SP204".SPARE_3,
                      signal06 := "SP204".SPARE_4,
                      signal07 := "SP204".SPARE_5,
                      interfaceSignals := "InstInterfaceSignals".statInterfaceSignalsHmi[63].valueSymbolLeft);
END_REGION

REGION Network 69: Interface Signals 64 SP 205
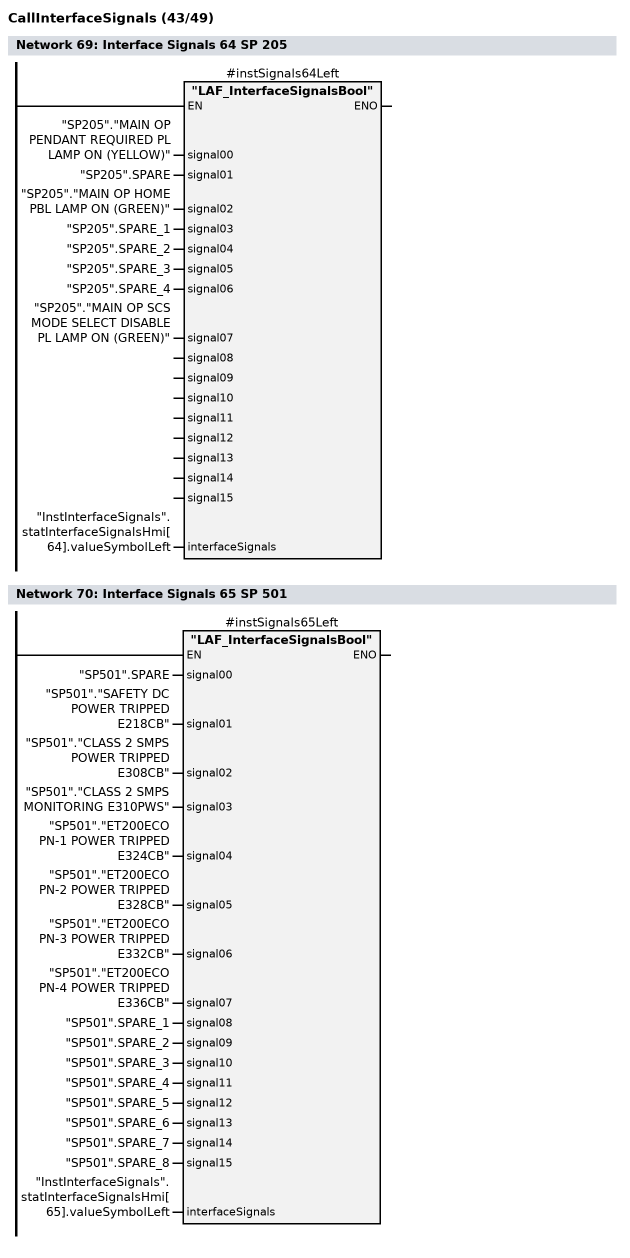
   RUNG wire#powerrail
      #instSignals64Left(signal00 := "SP205"."MAIN OP PENDANT REQUIRED PL LAMP ON (YELLOW)", signal01 := "SP205".SPARE, signal02 := "SP205"."MAIN OP HOME PBL LAMP ON (GREEN)", signal03 := "SP205".SPARE_1, signal04 := "SP205".SPARE_2, signal05 := "SP205".SPARE_3, signal06 := "SP205".SPARE_4, signal07 := "SP205"."MAIN OP SCS MODE SELECT DISABLE PL LAMP ON (GREEN)", signal08 :=, signal09 :=, signal10 :=, signal11 :=, signal12 :=, signal13 :=, signal14 :=, signal15 :=, interfaceSignals := "InstInterfaceSignals".statInterfaceSignalsHmi[64].valueSymbolLeft)
   END_RUNG
   // the same network as SCL:
   #instSignals64Left(signal00 := "SP205"."MAIN OP PENDANT REQUIRED PL LAMP ON (YELLOW)",   // "LAF_InterfaceSignalsBool"
                      signal01 := "SP205".SPARE,
                      signal02 := "SP205"."MAIN OP HOME PBL LAMP ON (GREEN)",
                      signal03 := "SP205".SPARE_1,
                      signal04 := "SP205".SPARE_2,
                      signal05 := "SP205".SPARE_3,
                      signal06 := "SP205".SPARE_4,
                      signal07 := "SP205"."MAIN OP SCS MODE SELECT DISABLE PL LAMP ON (GREEN)",
                      interfaceSignals := "InstInterfaceSignals".statInterfaceSignalsHmi[64].valueSymbolLeft);
END_REGION

REGION Network 70: Interface Signals 65 SP 501
   RUNG wire#powerrail
      #instSignals65Left(signal00 := "SP501".SPARE, signal01 := "SP501"."SAFETY DC POWER TRIPPED E218CB", signal02 := "SP501"."CLASS 2 SMPS POWER TRIPPED E308CB", signal03 := "SP501"."CLASS 2 SMPS MONITORING E310PWS", signal04 := "SP501"."ET200ECO PN-1 POWER TRIPPED E324CB", signal05 := "SP501"."ET200ECO PN-2 POWER TRIPPED E328CB", signal06 := "SP501"."ET200ECO PN-3 POWER TRIPPED E332CB", signal07 := "SP501"."ET200ECO PN-4 POWER TRIPPED E336CB", signal08 := "SP501".SPARE_1, signal09 := "SP501".SPARE_2, signal10 := "SP501".SPARE_3, signal11 := "SP501".SPARE_4, signal12 := "SP501".SPARE_5, signal13 := "SP501".SPARE_6, signal14 := "SP501".SPARE_7, signal15 := "SP501".SPARE_8, interfaceSignals := "InstInterfaceSignals".statInterfaceSignalsHmi[65].valueSymbolLeft)
   END_RUNG
   // the same network as SCL:
   #instSignals65Left(signal00 := "SP501".SPARE,   // "LAF_InterfaceSignalsBool"
                      signal01 := "SP501"."SAFETY DC POWER TRIPPED E218CB",
                      signal02 := "SP501"."CLASS 2 SMPS POWER TRIPPED E308CB",
                      signal03 := "SP501"."CLASS 2 SMPS MONITORING E310PWS",
                      signal04 := "SP501"."ET200ECO PN-1 POWER TRIPPED E324CB",
                      signal05 := "SP501"."ET200ECO PN-2 POWER TRIPPED E328CB",
                      signal06 := "SP501"."ET200ECO PN-3 POWER TRIPPED E332CB",
                      signal07 := "SP501"."ET200ECO PN-4 POWER TRIPPED E336CB",
                      signal08 := "SP501".SPARE_1,
                      signal09 := "SP501".SPARE_2,
                      signal10 := "SP501".SPARE_3,
                      signal11 := "SP501".SPARE_4,
                      signal12 := "SP501".SPARE_5,
                      signal13 := "SP501".SPARE_6,
                      signal14 := "SP501".SPARE_7,
                      signal15 := "SP501".SPARE_8,
                      interfaceSignals := "InstInterfaceSignals".statInterfaceSignalsHmi[65].valueSymbolLeft);
END_REGION

REGION Network 71: Interface Signals 66 SP 502
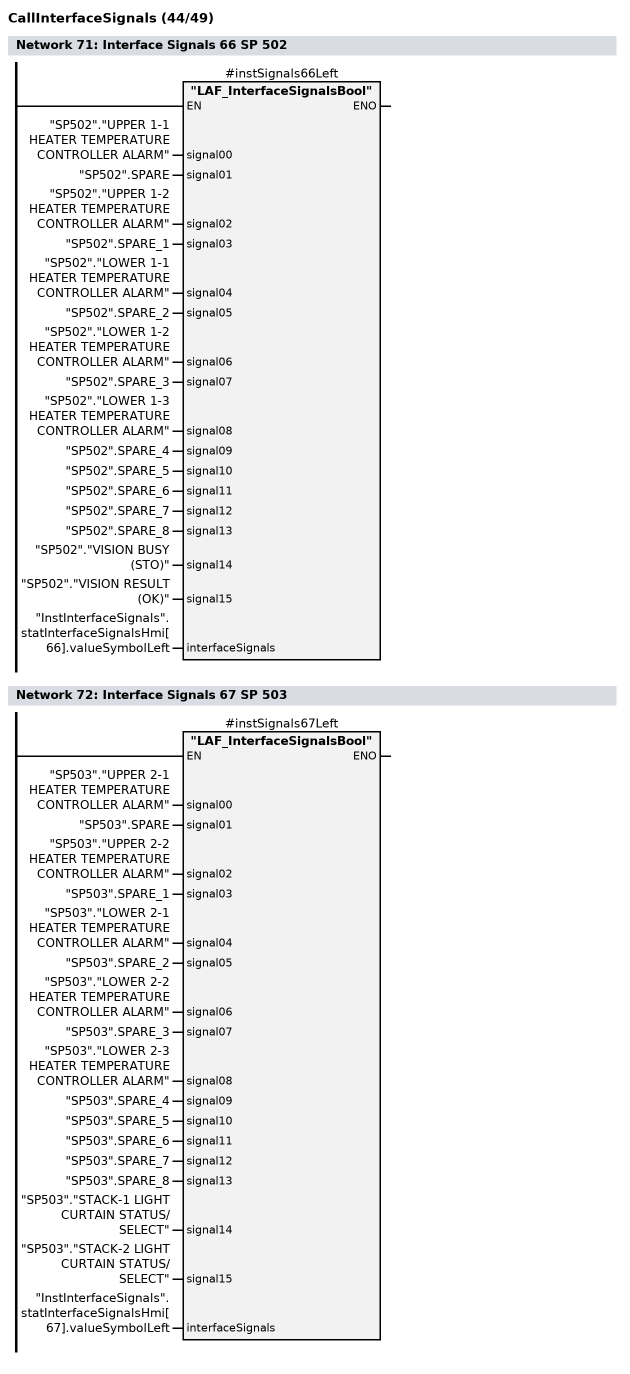
   RUNG wire#powerrail
      #instSignals66Left(signal00 := "SP502"."UPPER 1-1 HEATER TEMPERATURE CONTROLLER ALARM", signal01 := "SP502".SPARE, signal02 := "SP502"."UPPER 1-2 HEATER TEMPERATURE CONTROLLER ALARM", signal03 := "SP502".SPARE_1, signal04 := "SP502"."LOWER 1-1 HEATER TEMPERATURE CONTROLLER ALARM", signal05 := "SP502".SPARE_2, signal06 := "SP502"."LOWER 1-2 HEATER TEMPERATURE CONTROLLER ALARM", signal07 := "SP502".SPARE_3, signal08 := "SP502"."LOWER 1-3 HEATER TEMPERATURE CONTROLLER ALARM", signal09 := "SP502".SPARE_4, signal10 := "SP502".SPARE_5, signal11 := "SP502".SPARE_6, signal12 := "SP502".SPARE_7, signal13 := "SP502".SPARE_8, signal14 := "SP502"."VISION BUSY (STO)", signal15 := "SP502"."VISION RESULT (OK)", interfaceSignals := "InstInterfaceSignals".statInterfaceSignalsHmi[66].valueSymbolLeft)
   END_RUNG
   // the same network as SCL:
   #instSignals66Left(signal00 := "SP502"."UPPER 1-1 HEATER TEMPERATURE CONTROLLER ALARM",   // "LAF_InterfaceSignalsBool"
                      signal01 := "SP502".SPARE,
                      signal02 := "SP502"."UPPER 1-2 HEATER TEMPERATURE CONTROLLER ALARM",
                      signal03 := "SP502".SPARE_1,
                      signal04 := "SP502"."LOWER 1-1 HEATER TEMPERATURE CONTROLLER ALARM",
                      signal05 := "SP502".SPARE_2,
                      signal06 := "SP502"."LOWER 1-2 HEATER TEMPERATURE CONTROLLER ALARM",
                      signal07 := "SP502".SPARE_3,
                      signal08 := "SP502"."LOWER 1-3 HEATER TEMPERATURE CONTROLLER ALARM",
                      signal09 := "SP502".SPARE_4,
                      signal10 := "SP502".SPARE_5,
                      signal11 := "SP502".SPARE_6,
                      signal12 := "SP502".SPARE_7,
                      signal13 := "SP502".SPARE_8,
                      signal14 := "SP502"."VISION BUSY (STO)",
                      signal15 := "SP502"."VISION RESULT (OK)",
                      interfaceSignals := "InstInterfaceSignals".statInterfaceSignalsHmi[66].valueSymbolLeft);
END_REGION

REGION Network 72: Interface Signals 67 SP 503
   RUNG wire#powerrail
      #instSignals67Left(signal00 := "SP503"."UPPER 2-1 HEATER TEMPERATURE CONTROLLER ALARM", signal01 := "SP503".SPARE, signal02 := "SP503"."UPPER 2-2 HEATER TEMPERATURE CONTROLLER ALARM", signal03 := "SP503".SPARE_1, signal04 := "SP503"."LOWER 2-1 HEATER TEMPERATURE CONTROLLER ALARM", signal05 := "SP503".SPARE_2, signal06 := "SP503"."LOWER 2-2 HEATER TEMPERATURE CONTROLLER ALARM", signal07 := "SP503".SPARE_3, signal08 := "SP503"."LOWER 2-3 HEATER TEMPERATURE CONTROLLER ALARM", signal09 := "SP503".SPARE_4, signal10 := "SP503".SPARE_5, signal11 := "SP503".SPARE_6, signal12 := "SP503".SPARE_7, signal13 := "SP503".SPARE_8, signal14 := "SP503"."STACK-1 LIGHT CURTAIN STATUS/SELECT", signal15 := "SP503"."STACK-2 LIGHT CURTAIN STATUS/SELECT", interfaceSignals := "InstInterfaceSignals".statInterfaceSignalsHmi[67].valueSymbolLeft)
   END_RUNG
   // the same network as SCL:
   #instSignals67Left(signal00 := "SP503"."UPPER 2-1 HEATER TEMPERATURE CONTROLLER ALARM",   // "LAF_InterfaceSignalsBool"
                      signal01 := "SP503".SPARE,
                      signal02 := "SP503"."UPPER 2-2 HEATER TEMPERATURE CONTROLLER ALARM",
                      signal03 := "SP503".SPARE_1,
                      signal04 := "SP503"."LOWER 2-1 HEATER TEMPERATURE CONTROLLER ALARM",
                      signal05 := "SP503".SPARE_2,
                      signal06 := "SP503"."LOWER 2-2 HEATER TEMPERATURE CONTROLLER ALARM",
                      signal07 := "SP503".SPARE_3,
                      signal08 := "SP503"."LOWER 2-3 HEATER TEMPERATURE CONTROLLER ALARM",
                      signal09 := "SP503".SPARE_4,
                      signal10 := "SP503".SPARE_5,
                      signal11 := "SP503".SPARE_6,
                      signal12 := "SP503".SPARE_7,
                      signal13 := "SP503".SPARE_8,
                      signal14 := "SP503"."STACK-1 LIGHT CURTAIN STATUS/SELECT",
                      signal15 := "SP503"."STACK-2 LIGHT CURTAIN STATUS/SELECT",
                      interfaceSignals := "InstInterfaceSignals".statInterfaceSignalsHmi[67].valueSymbolLeft);
END_REGION

REGION Network 73: Interface Signals 68 SP 504
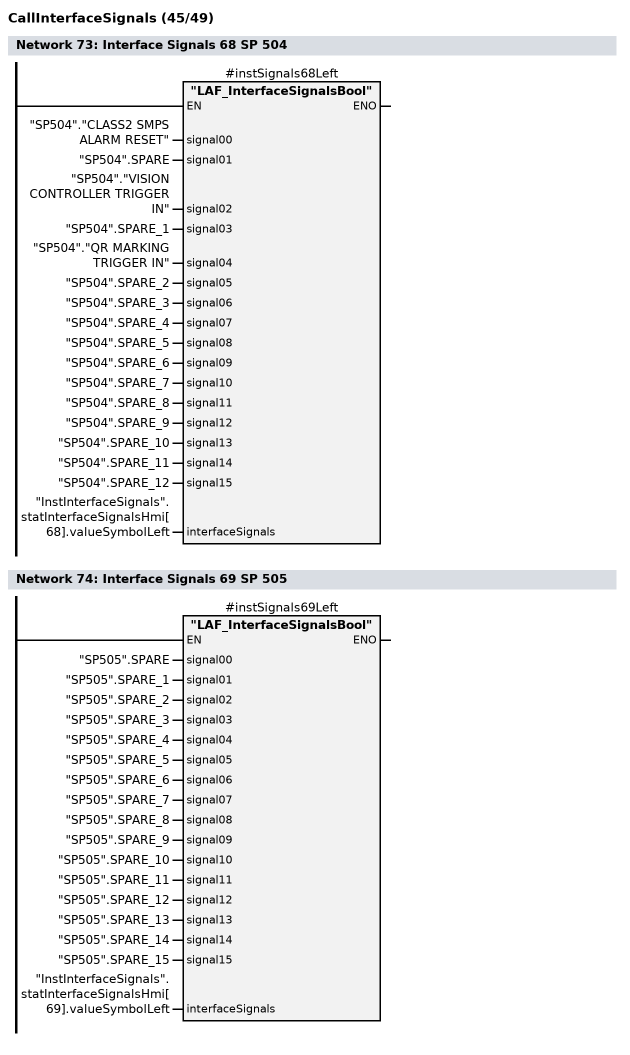
   RUNG wire#powerrail
      #instSignals68Left(signal00 := "SP504"."CLASS2 SMPS ALARM RESET", signal01 := "SP504".SPARE, signal02 := "SP504"."VISION CONTROLLER TRIGGER IN", signal03 := "SP504".SPARE_1, signal04 := "SP504"."QR MARKING TRIGGER IN", signal05 := "SP504".SPARE_2, signal06 := "SP504".SPARE_3, signal07 := "SP504".SPARE_4, signal08 := "SP504".SPARE_5, signal09 := "SP504".SPARE_6, signal10 := "SP504".SPARE_7, signal11 := "SP504".SPARE_8, signal12 := "SP504".SPARE_9, signal13 := "SP504".SPARE_10, signal14 := "SP504".SPARE_11, signal15 := "SP504".SPARE_12, interfaceSignals := "InstInterfaceSignals".statInterfaceSignalsHmi[68].valueSymbolLeft)
   END_RUNG
   // the same network as SCL:
   #instSignals68Left(signal00 := "SP504"."CLASS2 SMPS ALARM RESET",   // "LAF_InterfaceSignalsBool"
                      signal01 := "SP504".SPARE,
                      signal02 := "SP504"."VISION CONTROLLER TRIGGER IN",
                      signal03 := "SP504".SPARE_1,
                      signal04 := "SP504"."QR MARKING TRIGGER IN",
                      signal05 := "SP504".SPARE_2,
                      signal06 := "SP504".SPARE_3,
                      signal07 := "SP504".SPARE_4,
                      signal08 := "SP504".SPARE_5,
                      signal09 := "SP504".SPARE_6,
                      signal10 := "SP504".SPARE_7,
                      signal11 := "SP504".SPARE_8,
                      signal12 := "SP504".SPARE_9,
                      signal13 := "SP504".SPARE_10,
                      signal14 := "SP504".SPARE_11,
                      signal15 := "SP504".SPARE_12,
                      interfaceSignals := "InstInterfaceSignals".statInterfaceSignalsHmi[68].valueSymbolLeft);
END_REGION

REGION Network 74: Interface Signals 69 SP 505
   RUNG wire#powerrail
      #instSignals69Left(signal00 := "SP505".SPARE, signal01 := "SP505".SPARE_1, signal02 := "SP505".SPARE_2, signal03 := "SP505".SPARE_3, signal04 := "SP505".SPARE_4, signal05 := "SP505".SPARE_5, signal06 := "SP505".SPARE_6, signal07 := "SP505".SPARE_7, signal08 := "SP505".SPARE_8, signal09 := "SP505".SPARE_9, signal10 := "SP505".SPARE_10, signal11 := "SP505".SPARE_11, signal12 := "SP505".SPARE_12, signal13 := "SP505".SPARE_13, signal14 := "SP505".SPARE_14, signal15 := "SP505".SPARE_15, interfaceSignals := "InstInterfaceSignals".statInterfaceSignalsHmi[69].valueSymbolLeft)
   END_RUNG
   // the same network as SCL:
   #instSignals69Left(signal00 := "SP505".SPARE,   // "LAF_InterfaceSignalsBool"
                      signal01 := "SP505".SPARE_1,
                      signal02 := "SP505".SPARE_2,
                      signal03 := "SP505".SPARE_3,
                      signal04 := "SP505".SPARE_4,
                      signal05 := "SP505".SPARE_5,
                      signal06 := "SP505".SPARE_6,
                      signal07 := "SP505".SPARE_7,
                      signal08 := "SP505".SPARE_8,
                      signal09 := "SP505".SPARE_9,
                      signal10 := "SP505".SPARE_10,
                      signal11 := "SP505".SPARE_11,
                      signal12 := "SP505".SPARE_12,
                      signal13 := "SP505".SPARE_13,
                      signal14 := "SP505".SPARE_14,
                      signal15 := "SP505".SPARE_15,
                      interfaceSignals := "InstInterfaceSignals".statInterfaceSignalsHmi[69].valueSymbolLeft);
END_REGION

REGION Network 75: Interface Signals 70 SP 506
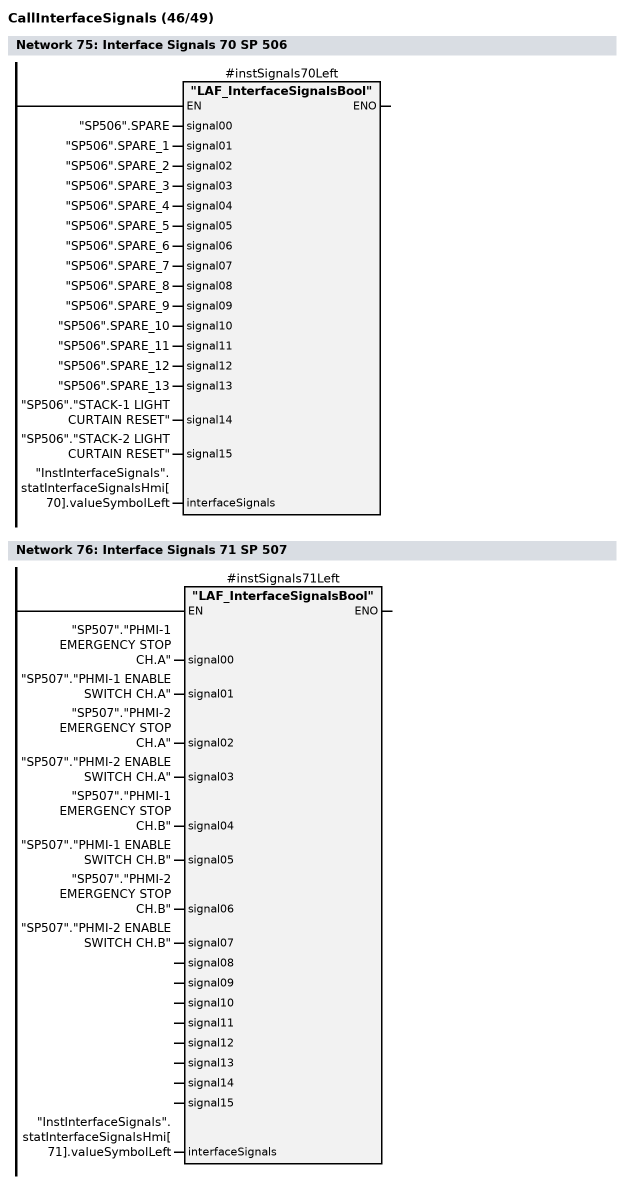
   RUNG wire#powerrail
      #instSignals70Left(signal00 := "SP506".SPARE, signal01 := "SP506".SPARE_1, signal02 := "SP506".SPARE_2, signal03 := "SP506".SPARE_3, signal04 := "SP506".SPARE_4, signal05 := "SP506".SPARE_5, signal06 := "SP506".SPARE_6, signal07 := "SP506".SPARE_7, signal08 := "SP506".SPARE_8, signal09 := "SP506".SPARE_9, signal10 := "SP506".SPARE_10, signal11 := "SP506".SPARE_11, signal12 := "SP506".SPARE_12, signal13 := "SP506".SPARE_13, signal14 := "SP506"."STACK-1 LIGHT CURTAIN RESET", signal15 := "SP506"."STACK-2 LIGHT CURTAIN RESET", interfaceSignals := "InstInterfaceSignals".statInterfaceSignalsHmi[70].valueSymbolLeft)
   END_RUNG
   // the same network as SCL:
   #instSignals70Left(signal00 := "SP506".SPARE,   // "LAF_InterfaceSignalsBool"
                      signal01 := "SP506".SPARE_1,
                      signal02 := "SP506".SPARE_2,
                      signal03 := "SP506".SPARE_3,
                      signal04 := "SP506".SPARE_4,
                      signal05 := "SP506".SPARE_5,
                      signal06 := "SP506".SPARE_6,
                      signal07 := "SP506".SPARE_7,
                      signal08 := "SP506".SPARE_8,
                      signal09 := "SP506".SPARE_9,
                      signal10 := "SP506".SPARE_10,
                      signal11 := "SP506".SPARE_11,
                      signal12 := "SP506".SPARE_12,
                      signal13 := "SP506".SPARE_13,
                      signal14 := "SP506"."STACK-1 LIGHT CURTAIN RESET",
                      signal15 := "SP506"."STACK-2 LIGHT CURTAIN RESET",
                      interfaceSignals := "InstInterfaceSignals".statInterfaceSignalsHmi[70].valueSymbolLeft);
END_REGION

REGION Network 76: Interface Signals 71 SP 507
   RUNG wire#powerrail
      #instSignals71Left(signal00 := "SP507"."PHMI-1 EMERGENCY STOP CH.A", signal01 := "SP507"."PHMI-1 ENABLE SWITCH CH.A", signal02 := "SP507"."PHMI-2 EMERGENCY STOP CH.A", signal03 := "SP507"."PHMI-2 ENABLE SWITCH CH.A", signal04 := "SP507"."PHMI-1 EMERGENCY STOP CH.B", signal05 := "SP507"."PHMI-1 ENABLE SWITCH CH.B", signal06 := "SP507"."PHMI-2 EMERGENCY STOP CH.B", signal07 := "SP507"."PHMI-2 ENABLE SWITCH CH.B", signal08 :=, signal09 :=, signal10 :=, signal11 :=, signal12 :=, signal13 :=, signal14 :=, signal15 :=, interfaceSignals := "InstInterfaceSignals".statInterfaceSignalsHmi[71].valueSymbolLeft)
   END_RUNG
   // the same network as SCL:
   #instSignals71Left(signal00 := "SP507"."PHMI-1 EMERGENCY STOP CH.A",   // "LAF_InterfaceSignalsBool"
                      signal01 := "SP507"."PHMI-1 ENABLE SWITCH CH.A",
                      signal02 := "SP507"."PHMI-2 EMERGENCY STOP CH.A",
                      signal03 := "SP507"."PHMI-2 ENABLE SWITCH CH.A",
                      signal04 := "SP507"."PHMI-1 EMERGENCY STOP CH.B",
                      signal05 := "SP507"."PHMI-1 ENABLE SWITCH CH.B",
                      signal06 := "SP507"."PHMI-2 EMERGENCY STOP CH.B",
                      signal07 := "SP507"."PHMI-2 ENABLE SWITCH CH.B",
                      interfaceSignals := "InstInterfaceSignals".statInterfaceSignalsHmi[71].valueSymbolLeft);
END_REGION

REGION Network 77: Interface Signals 72 SP 508
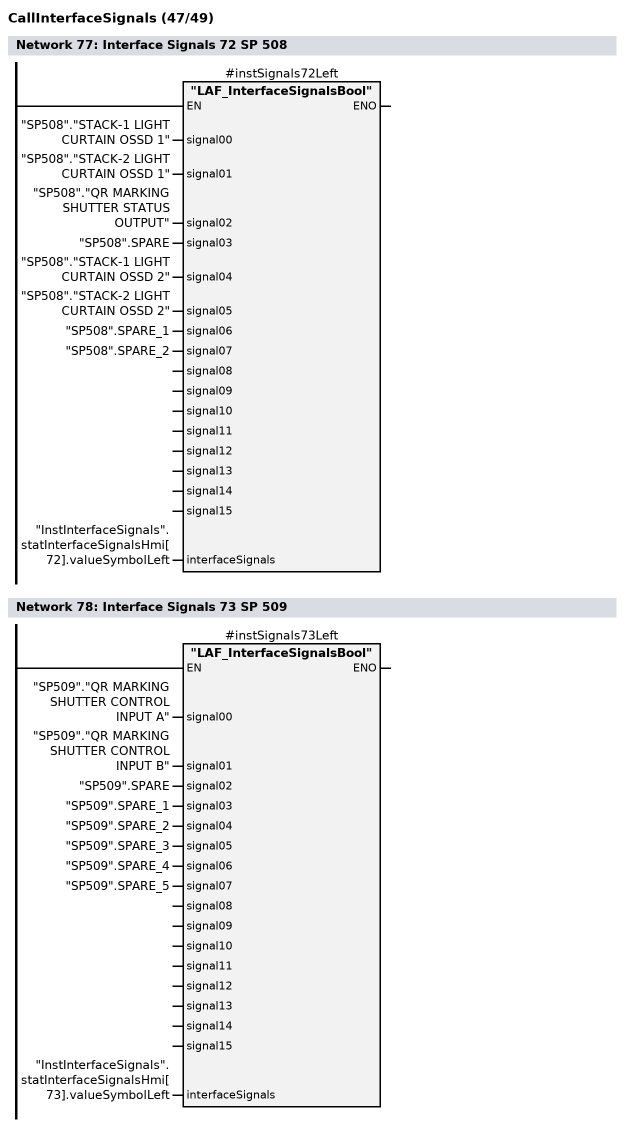
   RUNG wire#powerrail
      #instSignals72Left(signal00 := "SP508"."STACK-1 LIGHT CURTAIN OSSD 1", signal01 := "SP508"."STACK-2 LIGHT CURTAIN OSSD 1", signal02 := "SP508"."QR MARKING SHUTTER STATUS OUTPUT", signal03 := "SP508".SPARE, signal04 := "SP508"."STACK-1 LIGHT CURTAIN OSSD 2", signal05 := "SP508"."STACK-2 LIGHT CURTAIN OSSD 2", signal06 := "SP508".SPARE_1, signal07 := "SP508".SPARE_2, signal08 :=, signal09 :=, signal10 :=, signal11 :=, signal12 :=, signal13 :=, signal14 :=, signal15 :=, interfaceSignals := "InstInterfaceSignals".statInterfaceSignalsHmi[72].valueSymbolLeft)
   END_RUNG
   // the same network as SCL:
   #instSignals72Left(signal00 := "SP508"."STACK-1 LIGHT CURTAIN OSSD 1",   // "LAF_InterfaceSignalsBool"
                      signal01 := "SP508"."STACK-2 LIGHT CURTAIN OSSD 1",
                      signal02 := "SP508"."QR MARKING SHUTTER STATUS OUTPUT",
                      signal03 := "SP508".SPARE,
                      signal04 := "SP508"."STACK-1 LIGHT CURTAIN OSSD 2",
                      signal05 := "SP508"."STACK-2 LIGHT CURTAIN OSSD 2",
                      signal06 := "SP508".SPARE_1,
                      signal07 := "SP508".SPARE_2,
                      interfaceSignals := "InstInterfaceSignals".statInterfaceSignalsHmi[72].valueSymbolLeft);
END_REGION

REGION Network 78: Interface Signals 73 SP 509
   RUNG wire#powerrail
      #instSignals73Left(signal00 := "SP509"."QR MARKING SHUTTER CONTROL INPUT A", signal01 := "SP509"."QR MARKING SHUTTER CONTROL INPUT B", signal02 := "SP509".SPARE, signal03 := "SP509".SPARE_1, signal04 := "SP509".SPARE_2, signal05 := "SP509".SPARE_3, signal06 := "SP509".SPARE_4, signal07 := "SP509".SPARE_5, signal08 :=, signal09 :=, signal10 :=, signal11 :=, signal12 :=, signal13 :=, signal14 :=, signal15 :=, interfaceSignals := "InstInterfaceSignals".statInterfaceSignalsHmi[73].valueSymbolLeft)
   END_RUNG
   // the same network as SCL:
   #instSignals73Left(signal00 := "SP509"."QR MARKING SHUTTER CONTROL INPUT A",   // "LAF_InterfaceSignalsBool"
                      signal01 := "SP509"."QR MARKING SHUTTER CONTROL INPUT B",
                      signal02 := "SP509".SPARE,
                      signal03 := "SP509".SPARE_1,
                      signal04 := "SP509".SPARE_2,
                      signal05 := "SP509".SPARE_3,
                      signal06 := "SP509".SPARE_4,
                      signal07 := "SP509".SPARE_5,
                      interfaceSignals := "InstInterfaceSignals".statInterfaceSignalsHmi[73].valueSymbolLeft);
END_REGION

REGION Network 79: Interface Signals 74 SP 510
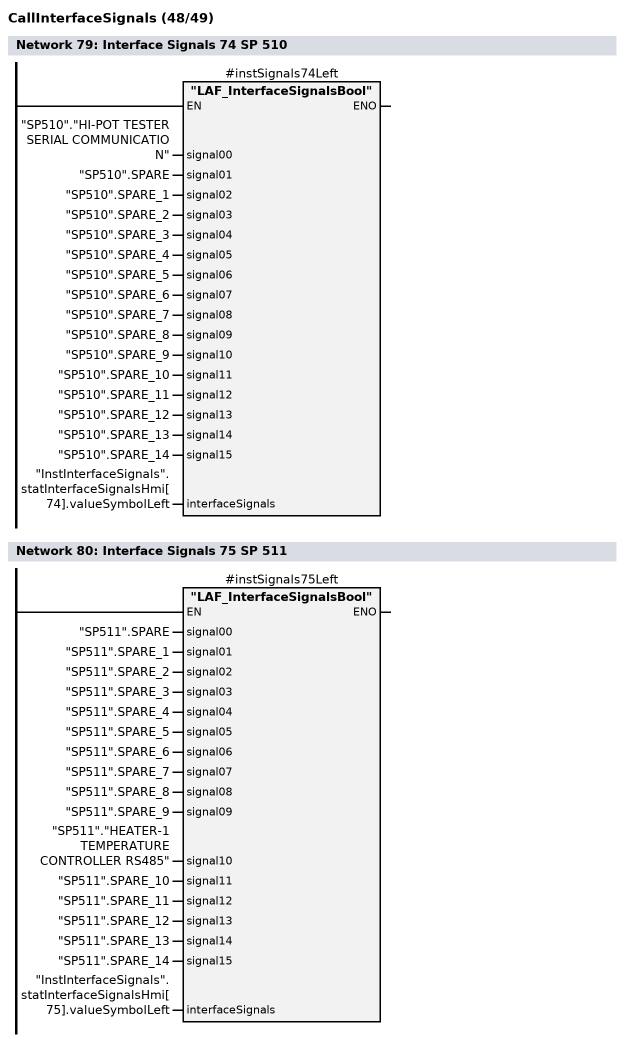
   RUNG wire#powerrail
      #instSignals74Left(signal00 := "SP510"."HI-POT TESTER SERIAL COMMUNICATION", signal01 := "SP510".SPARE, signal02 := "SP510".SPARE_1, signal03 := "SP510".SPARE_2, signal04 := "SP510".SPARE_3, signal05 := "SP510".SPARE_4, signal06 := "SP510".SPARE_5, signal07 := "SP510".SPARE_6, signal08 := "SP510".SPARE_7, signal09 := "SP510".SPARE_8, signal10 := "SP510".SPARE_9, signal11 := "SP510".SPARE_10, signal12 := "SP510".SPARE_11, signal13 := "SP510".SPARE_12, signal14 := "SP510".SPARE_13, signal15 := "SP510".SPARE_14, interfaceSignals := "InstInterfaceSignals".statInterfaceSignalsHmi[74].valueSymbolLeft)
   END_RUNG
   // the same network as SCL:
   #instSignals74Left(signal00 := "SP510"."HI-POT TESTER SERIAL COMMUNICATION",   // "LAF_InterfaceSignalsBool"
                      signal01 := "SP510".SPARE,
                      signal02 := "SP510".SPARE_1,
                      signal03 := "SP510".SPARE_2,
                      signal04 := "SP510".SPARE_3,
                      signal05 := "SP510".SPARE_4,
                      signal06 := "SP510".SPARE_5,
                      signal07 := "SP510".SPARE_6,
                      signal08 := "SP510".SPARE_7,
                      signal09 := "SP510".SPARE_8,
                      signal10 := "SP510".SPARE_9,
                      signal11 := "SP510".SPARE_10,
                      signal12 := "SP510".SPARE_11,
                      signal13 := "SP510".SPARE_12,
                      signal14 := "SP510".SPARE_13,
                      signal15 := "SP510".SPARE_14,
                      interfaceSignals := "InstInterfaceSignals".statInterfaceSignalsHmi[74].valueSymbolLeft);
END_REGION

REGION Network 80: Interface Signals 75 SP 511
   RUNG wire#powerrail
      #instSignals75Left(signal00 := "SP511".SPARE, signal01 := "SP511".SPARE_1, signal02 := "SP511".SPARE_2, signal03 := "SP511".SPARE_3, signal04 := "SP511".SPARE_4, signal05 := "SP511".SPARE_5, signal06 := "SP511".SPARE_6, signal07 := "SP511".SPARE_7, signal08 := "SP511".SPARE_8, signal09 := "SP511".SPARE_9, signal10 := "SP511"."HEATER-1 TEMPERATURE CONTROLLER RS485", signal11 := "SP511".SPARE_10, signal12 := "SP511".SPARE_11, signal13 := "SP511".SPARE_12, signal14 := "SP511".SPARE_13, signal15 := "SP511".SPARE_14, interfaceSignals := "InstInterfaceSignals".statInterfaceSignalsHmi[75].valueSymbolLeft)
   END_RUNG
   // the same network as SCL:
   #instSignals75Left(signal00 := "SP511".SPARE,   // "LAF_InterfaceSignalsBool"
                      signal01 := "SP511".SPARE_1,
                      signal02 := "SP511".SPARE_2,
                      signal03 := "SP511".SPARE_3,
                      signal04 := "SP511".SPARE_4,
                      signal05 := "SP511".SPARE_5,
                      signal06 := "SP511".SPARE_6,
                      signal07 := "SP511".SPARE_7,
                      signal08 := "SP511".SPARE_8,
                      signal09 := "SP511".SPARE_9,
                      signal10 := "SP511"."HEATER-1 TEMPERATURE CONTROLLER RS485",
                      signal11 := "SP511".SPARE_10,
                      signal12 := "SP511".SPARE_11,
                      signal13 := "SP511".SPARE_12,
                      signal14 := "SP511".SPARE_13,
                      signal15 := "SP511".SPARE_14,
                      interfaceSignals := "InstInterfaceSignals".statInterfaceSignalsHmi[75].valueSymbolLeft);
END_REGION

REGION Network 81: Interface Signals 76 SP 512
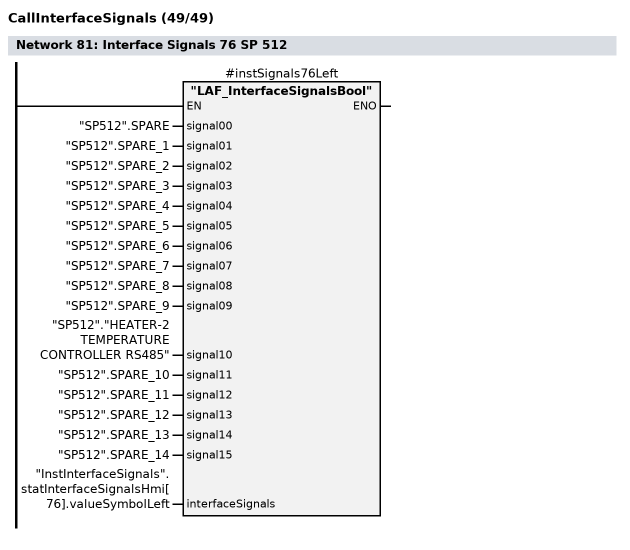
   RUNG wire#powerrail
      #instSignals76Left(signal00 := "SP512".SPARE, signal01 := "SP512".SPARE_1, signal02 := "SP512".SPARE_2, signal03 := "SP512".SPARE_3, signal04 := "SP512".SPARE_4, signal05 := "SP512".SPARE_5, signal06 := "SP512".SPARE_6, signal07 := "SP512".SPARE_7, signal08 := "SP512".SPARE_8, signal09 := "SP512".SPARE_9, signal10 := "SP512"."HEATER-2 TEMPERATURE CONTROLLER RS485", signal11 := "SP512".SPARE_10, signal12 := "SP512".SPARE_11, signal13 := "SP512".SPARE_12, signal14 := "SP512".SPARE_13, signal15 := "SP512".SPARE_14, interfaceSignals := "InstInterfaceSignals".statInterfaceSignalsHmi[76].valueSymbolLeft)
   END_RUNG
   // the same network as SCL:
   #instSignals76Left(signal00 := "SP512".SPARE,   // "LAF_InterfaceSignalsBool"
                      signal01 := "SP512".SPARE_1,
                      signal02 := "SP512".SPARE_2,
                      signal03 := "SP512".SPARE_3,
                      signal04 := "SP512".SPARE_4,
                      signal05 := "SP512".SPARE_5,
                      signal06 := "SP512".SPARE_6,
                      signal07 := "SP512".SPARE_7,
                      signal08 := "SP512".SPARE_8,
                      signal09 := "SP512".SPARE_9,
                      signal10 := "SP512"."HEATER-2 TEMPERATURE CONTROLLER RS485",
                      signal11 := "SP512".SPARE_10,
                      signal12 := "SP512".SPARE_11,
                      signal13 := "SP512".SPARE_12,
                      signal14 := "SP512".SPARE_13,
                      signal15 := "SP512".SPARE_14,
                      interfaceSignals := "InstInterfaceSignals".statInterfaceSignalsHmi[76].valueSymbolLeft);
END_REGION
END_FUNCTION_BLOCK

FUNCTION_BLOCK "CallInterfaceSignalsConv"   // FB213, LAD
// stored: MemoryReserve 100, SetENOAutomatically false
   VAR_INPUT
      InterfaceTestMode : Bool;
   END_VAR
   VAR_OUTPUT
      signals_I2S : "typeInspectionToStack";
      signals_S2I : "typeStackToInspection";
   END_VAR
   VAR_IN_OUT
      Comm_I2S : Array[0..95] of Bool;
      Comm_S2I : Array[0..95] of Bool;
      InterfaceTestButton : "LER_SignalsInput";
   END_VAR
   VAR
      statWordBuffer_I2S : Array[0..5] of Word;
      statWordBuffer_S2I : Array[0..5] of Word;
   END_VAR
   VAR_TEMP
      tempDeleteData : "LER_SignalsInput";
   END_VAR
   VAR CONSTANT
      TRUE : Bool := TRUE;
   END_VAR
   VAR_TEMP   // added for the SCL form of the ladder/FBD networks
      _w1 : Bool;
      _w2 : Bool;
      _w3 : Bool;
      _w4 : Bool;
   END_VAR
BEGIN

REGION Network 1: CommI2S -> signalsI2S
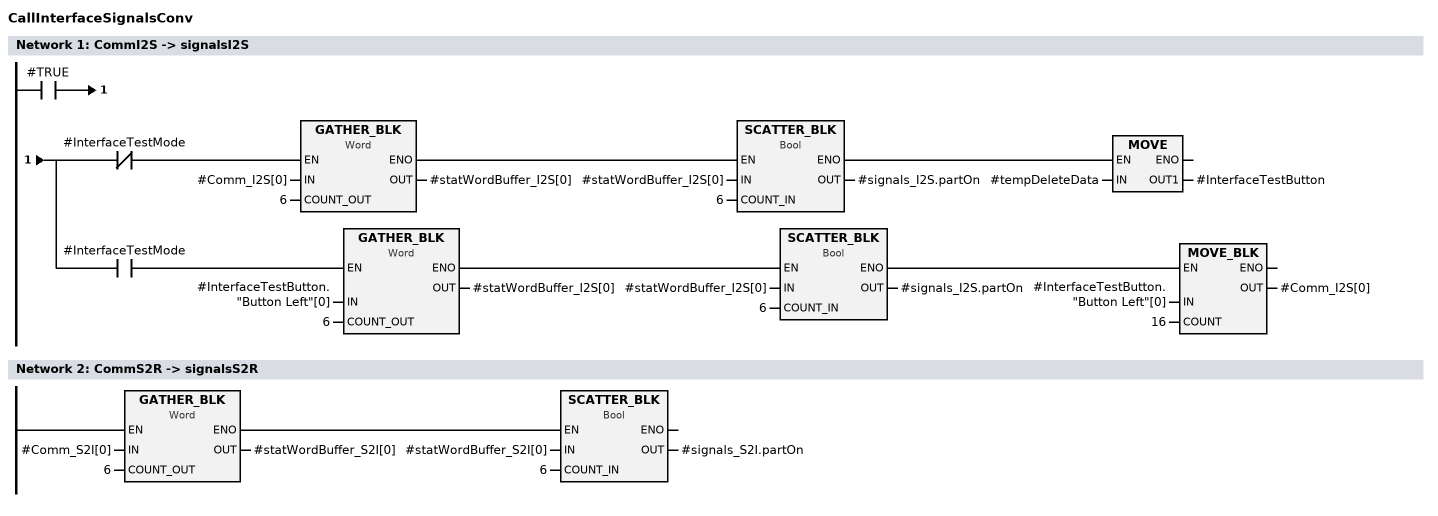
   GATHER_BLK(EN := #TRUE AND NOT #InterfaceTestMode,
              IN := #Comm_I2S[0],
              COUNT_OUT := 6,
              OUT => #statWordBuffer_I2S[0],
              ENO => #_w1);
   SCATTER_BLK(EN := #_w1, IN := #statWordBuffer_I2S[0], COUNT_IN := 6, OUT => #signals_I2S.partOn, ENO => #_w2);
   IF #_w2 THEN #InterfaceTestButton := #tempDeleteData; END_IF;
   GATHER_BLK(EN := #TRUE AND #InterfaceTestMode,
              IN := #InterfaceTestButton."Button Left"[0],
              COUNT_OUT := 6,
              OUT => #statWordBuffer_I2S[0],
              ENO => #_w3);
   SCATTER_BLK(EN := #_w3, IN := #statWordBuffer_I2S[0], COUNT_IN := 6, OUT => #signals_I2S.partOn, ENO => #_w4);
   IF #_w4 THEN
       MOVE_BLK(IN := #InterfaceTestButton."Button Left"[0], COUNT := 16, OUT => #Comm_I2S[0]);
   END_IF;
END_REGION

REGION Network 2: CommS2R -> signalsS2R
   RUNG wire#powerrail
      { S7_Templates := "[dest_type := Word, src_type := Bool, count_type := UInt]" } GATHER_BLK(IN := #Comm_S2I[0], COUNT_OUT := 6, OUT => #statWordBuffer_S2I[0])
      { S7_Templates := "[dest_type := Bool, src_type := Word, count_type := UInt]" } SCATTER_BLK(IN := #statWordBuffer_S2I[0], COUNT_IN := 6, OUT => #signals_S2I.partOn)
   END_RUNG
   // the same network as SCL:
   GATHER_BLK(IN := #Comm_S2I[0], COUNT_OUT := 6, OUT => #statWordBuffer_S2I[0], ENO => #_w1);
   IF #_w1 THEN SCATTER_BLK(IN := #statWordBuffer_S2I[0], COUNT_IN := 6, OUT => #signals_S2I.partOn); END_IF;
END_REGION
END_FUNCTION_BLOCK

FUNCTION_BLOCK "GetMotorstarterSignals"
{ S7_Optimized_Access := 'TRUE' ; Published := 'FALSE' }
VERSION : 0.1
   VAR_INPUT 
      Et200SpMotorstarterInterfaceAllUnits { ExternalAccessible := 'False'; ExternalVisible := 'False'; ExternalWritable := 'False'} : Array[1.."NO_OF_UNITS"] of "typeEmMotorStarterInterface";   // HMI: motorstarter values
      numberOfMS : USInt;
   END_VAR

   VAR_OUTPUT 
      selectedUnit : USInt;
      selectedEM : USInt;
      error : Word;
   END_VAR

   VAR_IN_OUT 
      Et200SpMotorstarterInterfaceHmi : "typeEt200SpMotorstarterInterfaceHmi";
   END_VAR

   VAR 
      statSelectedEMMotorStarter : USInt := 1;
      statSelectedUnitMotorStarter : USInt := 1;   // HMI: Selected unit
   END_VAR

   VAR_TEMP 
      tempEnable : Bool;   // Temporary value for input 'enable'
      tempEt200SpMotorstarterCurrent : Array[0.."NO_OF_ET200SPMOTORSTARTER"] of Real;
      tempEt200SpMotorstarterInputs : Array[0.."NO_OF_ET200SPMOTORSTARTER"] of "LSicar_typeMotorstarterIn";
      tempEt200SpMotorstarterOutputs : Array[0.."NO_OF_ET200SPMOTORSTARTER"] of "LSicar_typeMotorstarterOut";
      tempIndexMotorstarter : USInt;
      tempNoOfMS : USInt;
   END_VAR

   VAR CONSTANT 
      "INVALID UNIT" : Word := 16#7001;   // non existant unit
      "INVALID EM" : Word := 16#7002;   // non existant em
      OK : Word := 16#7000;
   END_VAR


BEGIN
	REGION BLOCK INFO HEADER
	    //===============================================================================
	    // Siemens AG / (c)Copyright 2024
	    //-------------------------------------------------------------------------------
	    // Title:            LAF_GetMotorstarterSignals
	    // Comment/Function: This block reads diagnostic information of a Motorstarter depending
	    //                   on the unit and Control Module selected in the HMI by the user.
	    // Library/Family:   Automation Framework / Motorstarter Diagnostic
	    // Author:           Siemens Digital Industries
	    // Tested with:      S7-1517TF V3.1
	    // Engineering:      TIA Portal V19
	    // Restrictions:     
	    //                   Required UDTs: LAF_typeDriveDiagConfig, LAF_typeDriveDiagInterfaceHmi
	    // Requirements:     S7-1500(T), MC_Version V8.0
	    //-------------------------------------------------------------------------------
	    // Change log table:
	    // Version  | Date       | Expert in charge        | Changes applied
	    //----------|------------|-------------------------|-----------------------------
	    // 01.00.00 | 05.06.2024 | SIMATIC Systems Support | First released version
	    //===============================================================================
	END_REGION BLOCK INFO HEADER
	
	REGION DESCRIPTION
	(/*
	This block reads diagnostic information (control inputs and outputs) of a Motorstarter. 
	At runtime, this block is enabled when the ET200SP Motorstarter screen is shown in the HMI. 
	Based on the selected motorstarter object in the HMI by the user. The shown information in the HMI depends on the
	Unit and Cotrol Module selected. 
	*/)
	END_REGION DESCRIPTION
	
	REGION INPUTS
	    //working with static values to keep the last selected value when opening for the first time the screen  
	  
	    #statSelectedUnitMotorStarter := #Et200SpMotorstarterInterfaceHmi.et200SpUnitMotorstarter;
	    #statSelectedEMMotorStarter := #Et200SpMotorstarterInterfaceHmi.et200SpEMMotorstarter;
	
	END_REGION INPUTS
	
	REGION ASSIGNING TEMPORARY VALUES
	    // Statement section REGION
	    IF #statSelectedUnitMotorStarter <= "NO_OF_UNITS" THEN
	        IF #statSelectedEMMotorStarter < "NO_OF_EM" THEN
	            #tempEt200SpMotorstarterCurrent := #Et200SpMotorstarterInterfaceAllUnits[#statSelectedUnitMotorStarter].EMmotorstarter[#statSelectedEMMotorStarter].et200SpMotorstarterCurrent;
	            #tempEt200SpMotorstarterInputs := #Et200SpMotorstarterInterfaceAllUnits[#statSelectedUnitMotorStarter].EMmotorstarter[#statSelectedEMMotorStarter].et200SpMotorstarterInputs;
	            #tempEt200SpMotorstarterOutputs := #Et200SpMotorstarterInterfaceAllUnits[#statSelectedUnitMotorStarter].EMmotorstarter[#statSelectedEMMotorStarter].et200SpMotorstarterOutputs;
	            #tempNoOfMS := #numberOfMS;
	            #error := #OK;
	        ELSE
	            #error := #"INVALID EM";
	        END_IF;
	
	    ELSE
	        #error := #"INVALID UNIT";
	    END_IF;
	
	
	END_REGION
	
	
	REGION OUTPUTS
	    // Statement section REGION
	    #Et200SpMotorstarterInterfaceHmi.et200SpMotorstarterCurrent := #tempEt200SpMotorstarterCurrent;
	    #Et200SpMotorstarterInterfaceHmi.et200SpMotorstarterInputs := #tempEt200SpMotorstarterInputs;
	    #Et200SpMotorstarterInterfaceHmi.et200SpMotorstarterOutputs := #tempEt200SpMotorstarterOutputs;
	    #Et200SpMotorstarterInterfaceHmi.et200SpNumberOfMotorstarters := #tempNoOfMS;
	    #selectedEM := #statSelectedEMMotorStarter;
	    #selectedUnit := #statSelectedUnitMotorStarter;
	END_REGION
	
	
END_FUNCTION_BLOCK

FUNCTION "DemoIdentRf" : Void   // FC39, LAD
TITLE = Demo: Ident
AUTHOR : SICAR
FAMILY : Demo
VERSION : 1.0
// Demo for usage of ident moduls
// stored: IsIECCheckEnabled true, SetENOAutomatically true
   // Ret_Val : Ret_Val
BEGIN

REGION Network 1: ChangeLog
   // Change log table:
   // Version | Date | Expert in charge | Changes applied
   // -------|---------|-------------|--------------------------------------------
   // 05.00.00 | 01.09.2023 | SICAR | First released version
END_REGION

REGION Network 2: Define reading informations
   // Write the String "Siemens" in the writting structur of the FB
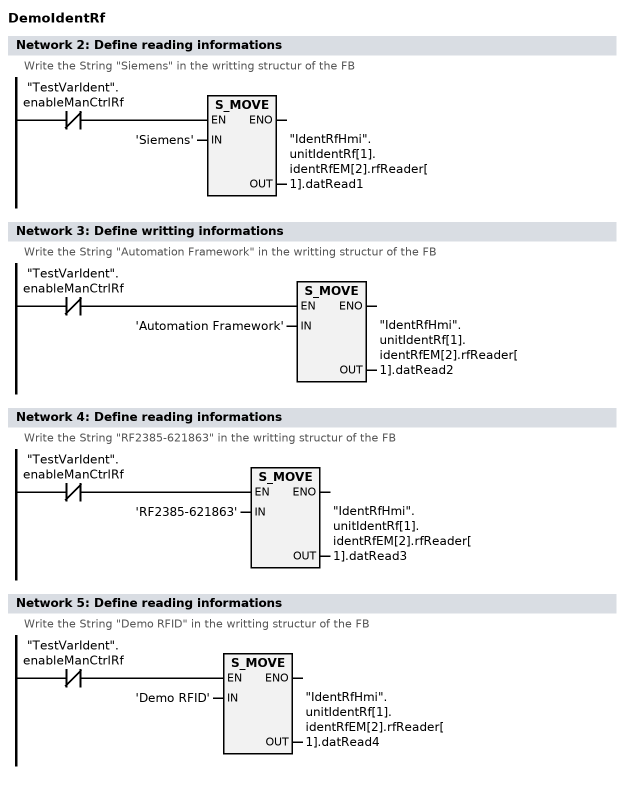
   RUNG wire#powerrail
      I_Contact( "TestVarIdent".enableManCtrlRf )
      S_Move(in := 'Siemens', out => "IdentRfHmi".unitIdentRf[1].identRfEM[2].rfReader[1].datRead1)
   END_RUNG
   // the same network as SCL:
   IF NOT "TestVarIdent".enableManCtrlRf THEN
       "IdentRfHmi".unitIdentRf[1].identRfEM[2].rfReader[1].datRead1 := 'Siemens';
   END_IF;
END_REGION

REGION Network 3: Define writting informations
   // Write the String "Automation Framework" in the writting structur of the FB
   RUNG wire#powerrail
      I_Contact( "TestVarIdent".enableManCtrlRf )
      S_Move(in := 'Automation Framework', out => "IdentRfHmi".unitIdentRf[1].identRfEM[2].rfReader[1].datRead2)
   END_RUNG
   // the same network as SCL:
   IF NOT "TestVarIdent".enableManCtrlRf THEN
       "IdentRfHmi".unitIdentRf[1].identRfEM[2].rfReader[1].datRead2 := 'Automation Framework';
   END_IF;
END_REGION

REGION Network 4: Define reading informations
   // Write the String "RF2385-621863" in the writting structur of the FB
   RUNG wire#powerrail
      I_Contact( "TestVarIdent".enableManCtrlRf )
      S_Move(in := 'RF2385-621863', out => "IdentRfHmi".unitIdentRf[1].identRfEM[2].rfReader[1].datRead3)
   END_RUNG
   // the same network as SCL:
   IF NOT "TestVarIdent".enableManCtrlRf THEN
       "IdentRfHmi".unitIdentRf[1].identRfEM[2].rfReader[1].datRead3 := 'RF2385-621863';
   END_IF;
END_REGION

REGION Network 5: Define reading informations
   // Write the String "Demo RFID" in the writting structur of the FB
   RUNG wire#powerrail
      I_Contact( "TestVarIdent".enableManCtrlRf )
      S_Move(in := 'Demo RFID', out => "IdentRfHmi".unitIdentRf[1].identRfEM[2].rfReader[1].datRead4)
   END_RUNG
   // the same network as SCL:
   IF NOT "TestVarIdent".enableManCtrlRf THEN
       "IdentRfHmi".unitIdentRf[1].identRfEM[2].rfReader[1].datRead4 := 'Demo RFID';
   END_IF;
END_REGION
END_FUNCTION

FUNCTION_BLOCK "GetIdentRf"
{ S7_Optimized_Access := 'TRUE' ; Published := 'TRUE' }
VERSION : 0.1
   VAR_INPUT 
      identRfAllUnits { ExternalAccessible := 'False'; ExternalVisible := 'False'; ExternalWritable := 'False'} : Array[1.."NO_OF_UNITS"] of "typeEMIdentRf";   // HMI: motorstarter values
      numberOfRfReaders : USInt;
   END_VAR

   VAR_OUTPUT 
      selectedUnit : USInt := 1;
      selectedEM : USInt;
      error : Word;
   END_VAR

   VAR_IN_OUT 
      IdentRfInterfaceHmi : "typeIdentRfHmi";
   END_VAR

   VAR 
      statSelectedEMIdentRf : USInt := 1;
      statSelectedUnitIdentRf : USInt := 1;   // HMI: Selected unit
   END_VAR

   VAR_TEMP 
      tempEnable : Bool;   // Temporary value for input 'enable'
      tempRfReader : Array[0.."NO_OF_RF_IDENT_DEVICES"] of "LSicar_typeIdentInterfaceHmi";
      tempIndexIdentRf : USInt;
      tempNoOfidertRf : USInt;
   END_VAR

   VAR CONSTANT 
      "INVALID UNIT" : Word := 16#7001;   // non existant unit
      "INVALID EM" : Word := 16#7002;   // non existant em
      OK : Word := 16#7000;
   END_VAR


BEGIN
	REGION BLOCK INFO HEADER
	    //===============================================================================
	    // Siemens AG / (c)Copyright 2024
	    //-------------------------------------------------------------------------------
	    // Title:            LAF_GetMotorstarterSignals
	    // Comment/Function: This block reads diagnostic information of a Motorstarter depending
	    //                   on the unit and Control Module selected in the HMI by the user.
	    // Library/Family:   Automation Framework / Motorstarter Diagnostic
	    // Author:           Siemens Digital Industries
	    // Tested with:      S7-1517TF V3.1
	    // Engineering:      TIA Portal V19
	    // Restrictions:     
	    //                   Required UDTs: LAF_typeDriveDiagConfig, LAF_typeDriveDiagInterfaceHmi
	    // Requirements:     S7-1500(T), MC_Version V8.0
	    //-------------------------------------------------------------------------------
	    // Change log table:
	    // Version  | Date       | Expert in charge        | Changes applied
	    //----------|------------|-------------------------|-----------------------------
	    // 01.00.00 | 05.06.2024 | SIMATIC Systems Support | First released version
	    //===============================================================================
	END_REGION BLOCK INFO HEADER
	
	REGION DESCRIPTION
	(/*
	This block reads diagnostic information (control inputs and outputs) of a Motorstarter. 
	At runtime, this block is enabled when the ET200SP Motorstarter screen is shown in the HMI. 
	Based on the selected motorstarter object in the HMI by the user. The shown information in the HMI depends on the
	Unit and Cotrol Module selected. 
	*/)
	END_REGION DESCRIPTION
	
	REGION INPUTS
	    //working with static values to keep the last selected value when opening for the first time the screen  
	  
	    #statSelectedUnitIdentRf := #IdentRfInterfaceHmi.selectedUnit;
	    #statSelectedEMIdentRf := #IdentRfInterfaceHmi.selectedEM;
	
	END_REGION INPUTS
	
	REGION ASSIGNING TEMPORARY VALUES
	    // Statement section REGION
	    IF #statSelectedUnitIdentRf <= "NO_OF_UNITS" THEN
	        IF #statSelectedEMIdentRf < "NO_OF_EM" THEN
	            #tempRfReader:= #identRfAllUnits[#statSelectedUnitIdentRf].identRfEM[#statSelectedEMIdentRf].rfReader;
	            #tempNoOfidertRf := #numberOfRfReaders;
	             #error := #OK;
	        ELSE
	            #error := #"INVALID EM";
	        END_IF;
	
	    ELSE
	        #error := #"INVALID UNIT";
	    END_IF;
	
	
	END_REGION
	
	
	REGION OUTPUTS
	    // Statement section REGION
	    #IdentRfInterfaceHmi.rfReader := #tempRfReader;
	    #selectedEM := #statSelectedEMIdentRf;
	    #selectedUnit := #statSelectedUnitIdentRf;
	END_REGION
	
	
END_FUNCTION_BLOCK

FUNCTION "DemoIdentMv" : Void   // FC69, LAD
TITLE = Demo: Ident
AUTHOR : SICAR
FAMILY : Demo
VERSION : 1.0
// Demo for usage of ident moduls
// stored: IsIECCheckEnabled true, SetENOAutomatically true
   // Ret_Val : Ret_Val
BEGIN

REGION Network 1: ChangeLog
   // Change log table:
   // Version | Date | Expert in charge | Changes applied
   // -------|---------|-------------|--------------------------------------------
   // 05.00.00 | 01.09.2023 | SICAR | First released version
END_REGION

REGION Network 2: Call: Ident MV
   // Demonstrate the call and function of an optical reader MV device
END_REGION

REGION Network 3: Define reading informations
   // Write the String "Siemens" in the writting structur of the FB
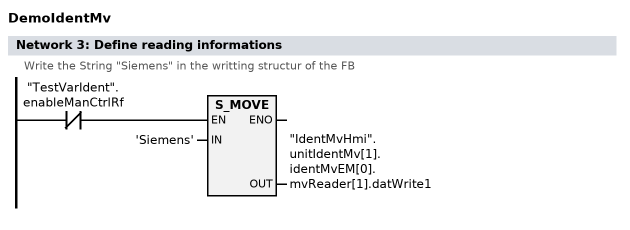
   RUNG wire#powerrail
      I_Contact( "TestVarIdent".enableManCtrlRf )
      S_Move(in := 'Siemens', out => "IdentMvHmi".unitIdentMv[1].identMvEM[0].mvReader[1].datWrite1)
   END_RUNG
   // the same network as SCL:
   IF NOT "TestVarIdent".enableManCtrlRf THEN
       "IdentMvHmi".unitIdentMv[1].identMvEM[0].mvReader[1].datWrite1 := 'Siemens';
   END_IF;
END_REGION
END_FUNCTION

FUNCTION_BLOCK "GetIdentMv"
{ S7_Optimized_Access := 'TRUE' ; Published := 'TRUE' }
VERSION : 0.1
   VAR_INPUT 
      identMvAllUnits { ExternalAccessible := 'False'; ExternalVisible := 'False'; ExternalWritable := 'False'} : Array[1.."NO_OF_UNITS"] of "typeEMIdentMv";   // HMI: motorstarter values
      numberOfMvReaders : USInt;
   END_VAR

   VAR_OUTPUT 
      selectedUnit : USInt;
      selectedEM : USInt;
      error : Word;
   END_VAR

   VAR_IN_OUT 
      IdentMvInterfaceHmi : "typeIdentMvHmi";
   END_VAR

   VAR 
      statSelectedEMIdentMv : USInt := 1;
      statSelectedUnitIdentRMv : USInt := 1;   // HMI: Selected unit
   END_VAR

   VAR_TEMP 
      tempEnable : Bool;   // Temporary value for input 'enable'
      tempMvReader : Array[0.."NO_OF_MV_IDENT_DEVICES"] of "LSicar_typeIdentInterfaceHmi";
      tempIndexIdentMv : USInt;
      tempNoOfidertMv : USInt;
   END_VAR

   VAR CONSTANT 
      "INVALID UNIT" : Word := 16#7001;   // non existant unit
      "INVALID EM" : Word := 16#7002;   // non existant em
      OK : Word := 16#7000;
   END_VAR


BEGIN
	REGION BLOCK INFO HEADER
	    //===============================================================================
	    // Siemens AG / (c)Copyright 2024
	    //-------------------------------------------------------------------------------
	    // Title:            LAF_GetMotorstarterSignals
	    // Comment/Function: This block reads diagnostic information of a Motorstarter depending
	    //                   on the unit and Control Module selected in the HMI by the user.
	    // Library/Family:   Automation Framework / Motorstarter Diagnostic
	    // Author:           Siemens Digital Industries
	    // Tested with:      S7-1517TF V3.1
	    // Engineering:      TIA Portal V19
	    // Restrictions:     
	    //                   Required UDTs: LAF_typeDriveDiagConfig, LAF_typeDriveDiagInterfaceHmi
	    // Requirements:     S7-1500(T), MC_Version V8.0
	    //-------------------------------------------------------------------------------
	    // Change log table:
	    // Version  | Date       | Expert in charge        | Changes applied
	    //----------|------------|-------------------------|-----------------------------
	    // 01.00.00 | 05.06.2024 | SIMATIC Systems Support | First released version
	    //===============================================================================
	END_REGION BLOCK INFO HEADER
	
	REGION DESCRIPTION
	(/*
	This block reads diagnostic information (control inputs and outputs) of a Motorstarter. 
	At runtime, this block is enabled when the ET200SP Motorstarter screen is shown in the HMI. 
	Based on the selected motorstarter object in the HMI by the user. The shown information in the HMI depends on the
	Unit and Cotrol Module selected. 
	*/)
	END_REGION DESCRIPTION
	
	REGION INPUTS
	    //working with static values to keep the last selected value when opening for the first time the screen  
	  
	    #statSelectedUnitIdentRMv := #IdentMvInterfaceHmi.selectedUnit;
	    #statSelectedEMIdentMv := #IdentMvInterfaceHmi.selectedEM;
	
	END_REGION INPUTS
	
	REGION ASSIGNING TEMPORARY VALUES
	    // Statement section REGION
	    IF #statSelectedUnitIdentRMv <= "NO_OF_UNITS" THEN
	        IF #statSelectedEMIdentMv < "NO_OF_EM" THEN
	            #tempMvReader := #identMvAllUnits[#statSelectedUnitIdentRMv].identMvEM[#statSelectedEMIdentMv].mvReader;
	            #tempNoOfidertMv := #numberOfMvReaders;
	            #error := #OK;
	        ELSE
	            #error := #"INVALID EM";
	        END_IF;
	
	    ELSE
	        #error := #"INVALID UNIT";
	    END_IF;
	
	
	END_REGION
	
	
	REGION OUTPUTS
	    // Statement section REGION
	    #IdentMvInterfaceHmi.mvReader := #tempMvReader;
	    #selectedEM := #statSelectedEMIdentMv;
	    #selectedUnit := #statSelectedUnitIdentRMv;
	END_REGION
	
	
END_FUNCTION_BLOCK

FUNCTION "SafetyDoor" : Void   // FC97, LAD
// stored: SetENOAutomatically false
   VAR CONSTANT
      TRUE : Bool := TRUE;
      FALSE : Bool;
   END_VAR
   VAR_TEMP   // added for the SCL form of the ladder/FBD networks
      _w1 : Bool;
   END_VAR
BEGIN

REGION Network 1: fDoor1 monitoring
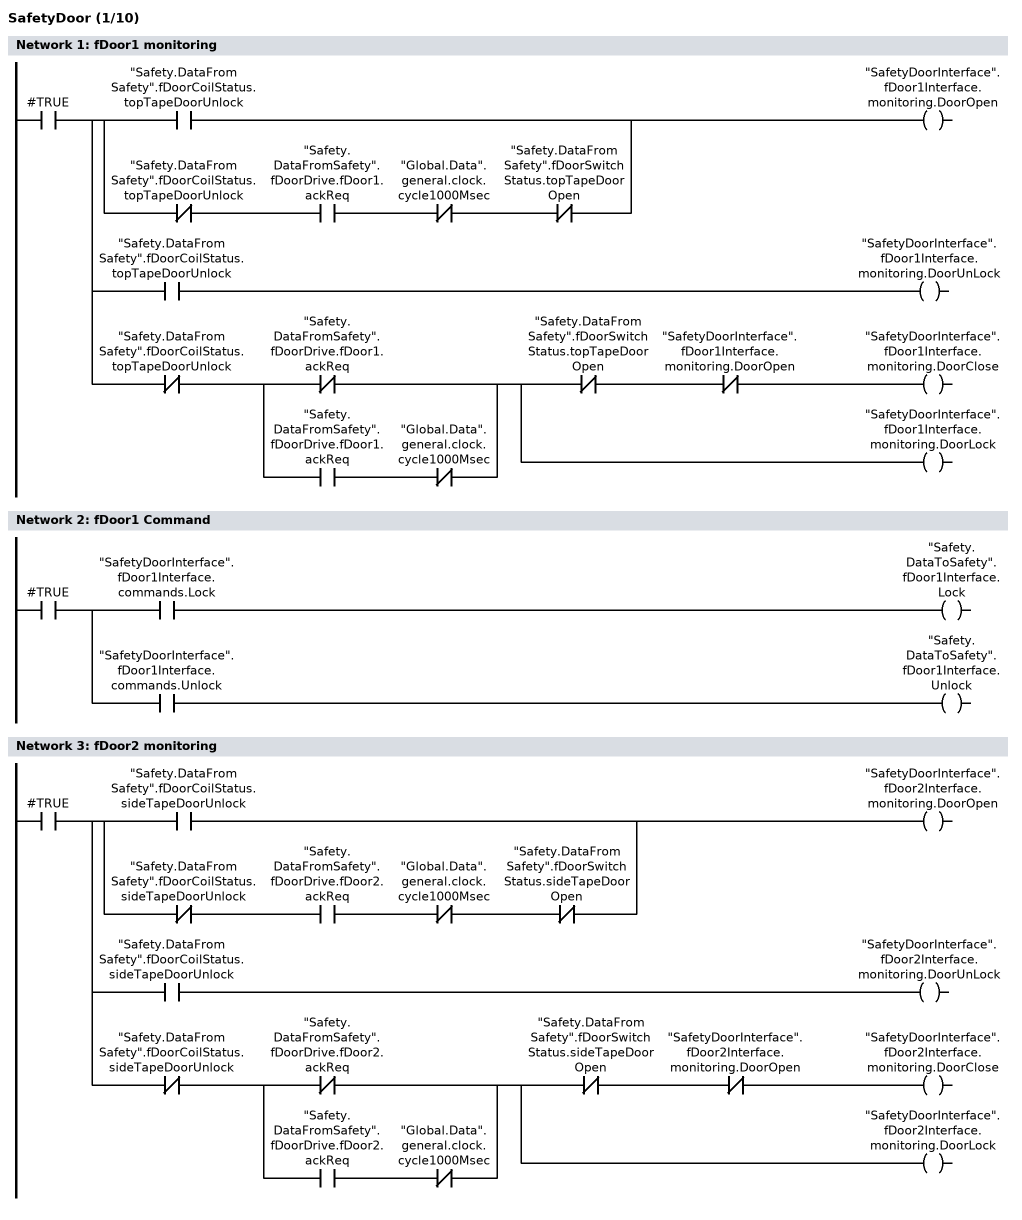
   RUNG wire#powerrail
      Contact( #TRUE )
      wire#w1
      Contact( "Safety.DataFromSafety".fDoorCoilStatus.topTapeDoorUnlock )
      wire#w2
      Coil( "SafetyDoorInterface".fDoor1Interface.monitoring.DoorOpen )
   END_RUNG
   RUNG wire#w1
      I_Contact( "Safety.DataFromSafety".fDoorCoilStatus.topTapeDoorUnlock )
      Contact( "Safety.DataFromSafety".fDoorDrive.fDoor1.ackReq )
      I_Contact( "Global.Data".general.clock.cycle1000Msec )
      I_Contact( "Safety.DataFromSafety".fDoorSwitchStatus.topTapeDoorOpen )
   END_RUNG wire#w2
   RUNG wire#w1
      Contact( "Safety.DataFromSafety".fDoorCoilStatus.topTapeDoorUnlock )
      Coil( "SafetyDoorInterface".fDoor1Interface.monitoring.DoorUnLock )
   END_RUNG
   RUNG wire#w1
      I_Contact( "Safety.DataFromSafety".fDoorCoilStatus.topTapeDoorUnlock )
      wire#w3
      I_Contact( "Safety.DataFromSafety".fDoorDrive.fDoor1.ackReq )
      wire#w4
      I_Contact( "Safety.DataFromSafety".fDoorSwitchStatus.topTapeDoorOpen )
      I_Contact( "SafetyDoorInterface".fDoor1Interface.monitoring.DoorOpen )
      Coil( "SafetyDoorInterface".fDoor1Interface.monitoring.DoorClose )
   END_RUNG
   RUNG wire#w3
      Contact( "Safety.DataFromSafety".fDoorDrive.fDoor1.ackReq )
      I_Contact( "Global.Data".general.clock.cycle1000Msec )
   END_RUNG wire#w4
   RUNG wire#w4
      Coil( "SafetyDoorInterface".fDoor1Interface.monitoring.DoorLock )
   END_RUNG
   // the same network as SCL:
   "SafetyDoorInterface".fDoor1Interface.monitoring.DoorOpen := #TRUE AND ("Safety.DataFromSafety".fDoorCoilStatus.topTapeDoorUnlock OR (NOT "Safety.DataFromSafety".fDoorCoilStatus.topTapeDoorUnlock AND "Safety.DataFromSafety".fDoorDrive.fDoor1.ackReq AND NOT "Global.Data".general.clock.cycle1000Msec AND NOT "Safety.DataFromSafety".fDoorSwitchStatus.topTapeDoorOpen));
   "SafetyDoorInterface".fDoor1Interface.monitoring.DoorUnLock := #TRUE AND "Safety.DataFromSafety".fDoorCoilStatus.topTapeDoorUnlock;
   #_w1 := #TRUE AND NOT "Safety.DataFromSafety".fDoorCoilStatus.topTapeDoorUnlock AND (NOT "Safety.DataFromSafety".fDoorDrive.fDoor1.ackReq OR ("Safety.DataFromSafety".fDoorDrive.fDoor1.ackReq AND NOT "Global.Data".general.clock.cycle1000Msec));
   "SafetyDoorInterface".fDoor1Interface.monitoring.DoorClose := #_w1 AND NOT "Safety.DataFromSafety".fDoorSwitchStatus.topTapeDoorOpen AND NOT "SafetyDoorInterface".fDoor1Interface.monitoring.DoorOpen;
   "SafetyDoorInterface".fDoor1Interface.monitoring.DoorLock := #_w1;
END_REGION

REGION Network 2: fDoor1 Command
   RUNG wire#powerrail
      Contact( #TRUE )
      wire#w1
      Contact( "SafetyDoorInterface".fDoor1Interface.commands.Lock )
      Coil( "Safety.DataToSafety".fDoor1Interface.Lock )
   END_RUNG
   RUNG wire#w1
      Contact( "SafetyDoorInterface".fDoor1Interface.commands.Unlock )
      Coil( "Safety.DataToSafety".fDoor1Interface.Unlock )
   END_RUNG
   // the same network as SCL:
   "Safety.DataToSafety".fDoor1Interface.Lock := #TRUE AND "SafetyDoorInterface".fDoor1Interface.commands.Lock;
   "Safety.DataToSafety".fDoor1Interface.Unlock := #TRUE AND "SafetyDoorInterface".fDoor1Interface.commands.Unlock;
END_REGION

REGION Network 3: fDoor2 monitoring
   RUNG wire#powerrail
      Contact( #TRUE )
      wire#w1
      Contact( "Safety.DataFromSafety".fDoorCoilStatus.sideTapeDoorUnlock )
      wire#w2
      Coil( "SafetyDoorInterface".fDoor2Interface.monitoring.DoorOpen )
   END_RUNG
   RUNG wire#w1
      I_Contact( "Safety.DataFromSafety".fDoorCoilStatus.sideTapeDoorUnlock )
      Contact( "Safety.DataFromSafety".fDoorDrive.fDoor2.ackReq )
      I_Contact( "Global.Data".general.clock.cycle1000Msec )
      I_Contact( "Safety.DataFromSafety".fDoorSwitchStatus.sideTapeDoorOpen )
   END_RUNG wire#w2
   RUNG wire#w1
      Contact( "Safety.DataFromSafety".fDoorCoilStatus.sideTapeDoorUnlock )
      Coil( "SafetyDoorInterface".fDoor2Interface.monitoring.DoorUnLock )
   END_RUNG
   RUNG wire#w1
      I_Contact( "Safety.DataFromSafety".fDoorCoilStatus.sideTapeDoorUnlock )
      wire#w3
      I_Contact( "Safety.DataFromSafety".fDoorDrive.fDoor2.ackReq )
      wire#w4
      I_Contact( "Safety.DataFromSafety".fDoorSwitchStatus.sideTapeDoorOpen )
      I_Contact( "SafetyDoorInterface".fDoor2Interface.monitoring.DoorOpen )
      Coil( "SafetyDoorInterface".fDoor2Interface.monitoring.DoorClose )
   END_RUNG
   RUNG wire#w3
      Contact( "Safety.DataFromSafety".fDoorDrive.fDoor2.ackReq )
      I_Contact( "Global.Data".general.clock.cycle1000Msec )
   END_RUNG wire#w4
   RUNG wire#w4
      Coil( "SafetyDoorInterface".fDoor2Interface.monitoring.DoorLock )
   END_RUNG
   // the same network as SCL:
   "SafetyDoorInterface".fDoor2Interface.monitoring.DoorOpen := #TRUE AND ("Safety.DataFromSafety".fDoorCoilStatus.sideTapeDoorUnlock OR (NOT "Safety.DataFromSafety".fDoorCoilStatus.sideTapeDoorUnlock AND "Safety.DataFromSafety".fDoorDrive.fDoor2.ackReq AND NOT "Global.Data".general.clock.cycle1000Msec AND NOT "Safety.DataFromSafety".fDoorSwitchStatus.sideTapeDoorOpen));
   "SafetyDoorInterface".fDoor2Interface.monitoring.DoorUnLock := #TRUE AND "Safety.DataFromSafety".fDoorCoilStatus.sideTapeDoorUnlock;
   #_w1 := #TRUE AND NOT "Safety.DataFromSafety".fDoorCoilStatus.sideTapeDoorUnlock AND (NOT "Safety.DataFromSafety".fDoorDrive.fDoor2.ackReq OR ("Safety.DataFromSafety".fDoorDrive.fDoor2.ackReq AND NOT "Global.Data".general.clock.cycle1000Msec));
   "SafetyDoorInterface".fDoor2Interface.monitoring.DoorClose := #_w1 AND NOT "Safety.DataFromSafety".fDoorSwitchStatus.sideTapeDoorOpen AND NOT "SafetyDoorInterface".fDoor2Interface.monitoring.DoorOpen;
   "SafetyDoorInterface".fDoor2Interface.monitoring.DoorLock := #_w1;
END_REGION

REGION Network 4: fDoor2 Command
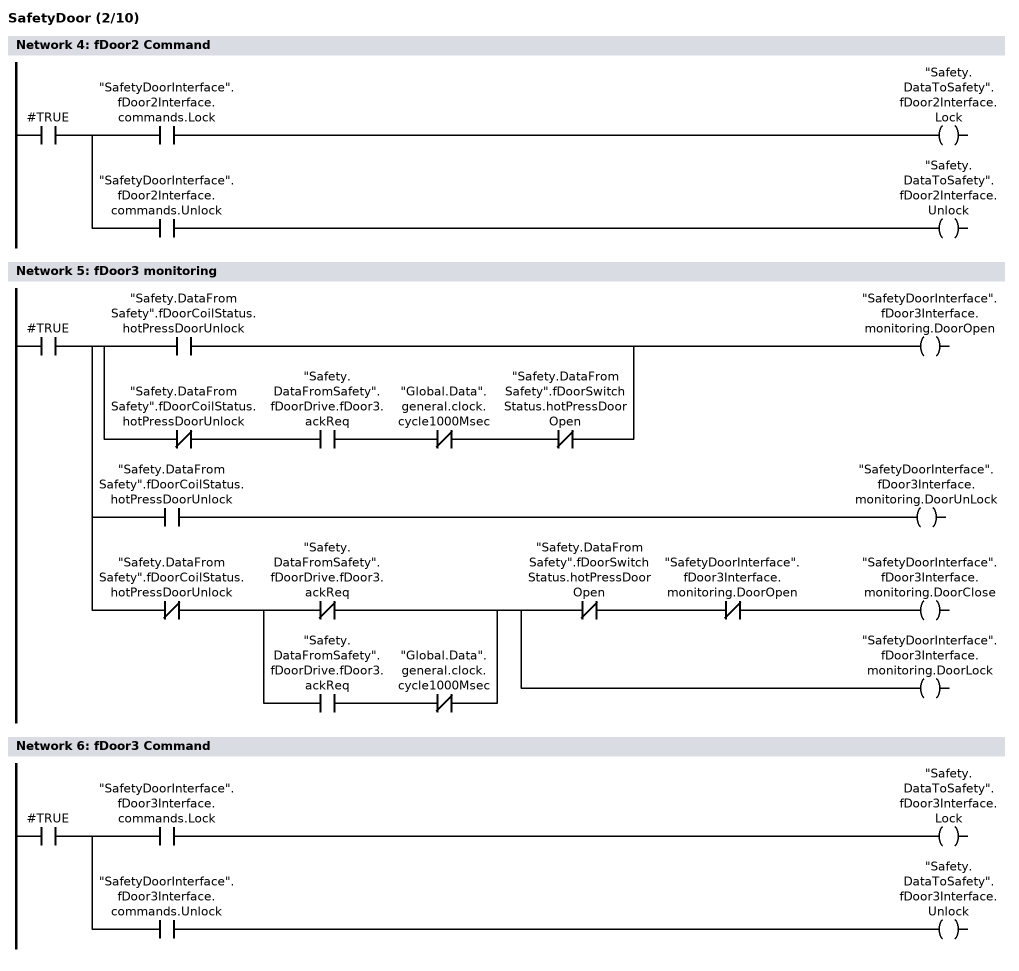
   RUNG wire#powerrail
      Contact( #TRUE )
      wire#w1
      Contact( "SafetyDoorInterface".fDoor2Interface.commands.Lock )
      Coil( "Safety.DataToSafety".fDoor2Interface.Lock )
   END_RUNG
   RUNG wire#w1
      Contact( "SafetyDoorInterface".fDoor2Interface.commands.Unlock )
      Coil( "Safety.DataToSafety".fDoor2Interface.Unlock )
   END_RUNG
   // the same network as SCL:
   "Safety.DataToSafety".fDoor2Interface.Lock := #TRUE AND "SafetyDoorInterface".fDoor2Interface.commands.Lock;
   "Safety.DataToSafety".fDoor2Interface.Unlock := #TRUE AND "SafetyDoorInterface".fDoor2Interface.commands.Unlock;
END_REGION

REGION Network 5: fDoor3 monitoring
   RUNG wire#powerrail
      Contact( #TRUE )
      wire#w1
      Contact( "Safety.DataFromSafety".fDoorCoilStatus.hotPressDoorUnlock )
      wire#w2
      Coil( "SafetyDoorInterface".fDoor3Interface.monitoring.DoorOpen )
   END_RUNG
   RUNG wire#w1
      I_Contact( "Safety.DataFromSafety".fDoorCoilStatus.hotPressDoorUnlock )
      Contact( "Safety.DataFromSafety".fDoorDrive.fDoor3.ackReq )
      I_Contact( "Global.Data".general.clock.cycle1000Msec )
      I_Contact( "Safety.DataFromSafety".fDoorSwitchStatus.hotPressDoorOpen )
   END_RUNG wire#w2
   RUNG wire#w1
      Contact( "Safety.DataFromSafety".fDoorCoilStatus.hotPressDoorUnlock )
      Coil( "SafetyDoorInterface".fDoor3Interface.monitoring.DoorUnLock )
   END_RUNG
   RUNG wire#w1
      I_Contact( "Safety.DataFromSafety".fDoorCoilStatus.hotPressDoorUnlock )
      wire#w3
      I_Contact( "Safety.DataFromSafety".fDoorDrive.fDoor3.ackReq )
      wire#w4
      I_Contact( "Safety.DataFromSafety".fDoorSwitchStatus.hotPressDoorOpen )
      I_Contact( "SafetyDoorInterface".fDoor3Interface.monitoring.DoorOpen )
      Coil( "SafetyDoorInterface".fDoor3Interface.monitoring.DoorClose )
   END_RUNG
   RUNG wire#w3
      Contact( "Safety.DataFromSafety".fDoorDrive.fDoor3.ackReq )
      I_Contact( "Global.Data".general.clock.cycle1000Msec )
   END_RUNG wire#w4
   RUNG wire#w4
      Coil( "SafetyDoorInterface".fDoor3Interface.monitoring.DoorLock )
   END_RUNG
   // the same network as SCL:
   "SafetyDoorInterface".fDoor3Interface.monitoring.DoorOpen := #TRUE AND ("Safety.DataFromSafety".fDoorCoilStatus.hotPressDoorUnlock OR (NOT "Safety.DataFromSafety".fDoorCoilStatus.hotPressDoorUnlock AND "Safety.DataFromSafety".fDoorDrive.fDoor3.ackReq AND NOT "Global.Data".general.clock.cycle1000Msec AND NOT "Safety.DataFromSafety".fDoorSwitchStatus.hotPressDoorOpen));
   "SafetyDoorInterface".fDoor3Interface.monitoring.DoorUnLock := #TRUE AND "Safety.DataFromSafety".fDoorCoilStatus.hotPressDoorUnlock;
   #_w1 := #TRUE AND NOT "Safety.DataFromSafety".fDoorCoilStatus.hotPressDoorUnlock AND (NOT "Safety.DataFromSafety".fDoorDrive.fDoor3.ackReq OR ("Safety.DataFromSafety".fDoorDrive.fDoor3.ackReq AND NOT "Global.Data".general.clock.cycle1000Msec));
   "SafetyDoorInterface".fDoor3Interface.monitoring.DoorClose := #_w1 AND NOT "Safety.DataFromSafety".fDoorSwitchStatus.hotPressDoorOpen AND NOT "SafetyDoorInterface".fDoor3Interface.monitoring.DoorOpen;
   "SafetyDoorInterface".fDoor3Interface.monitoring.DoorLock := #_w1;
END_REGION

REGION Network 6: fDoor3 Command
   RUNG wire#powerrail
      Contact( #TRUE )
      wire#w1
      Contact( "SafetyDoorInterface".fDoor3Interface.commands.Lock )
      Coil( "Safety.DataToSafety".fDoor3Interface.Lock )
   END_RUNG
   RUNG wire#w1
      Contact( "SafetyDoorInterface".fDoor3Interface.commands.Unlock )
      Coil( "Safety.DataToSafety".fDoor3Interface.Unlock )
   END_RUNG
   // the same network as SCL:
   "Safety.DataToSafety".fDoor3Interface.Lock := #TRUE AND "SafetyDoorInterface".fDoor3Interface.commands.Lock;
   "Safety.DataToSafety".fDoor3Interface.Unlock := #TRUE AND "SafetyDoorInterface".fDoor3Interface.commands.Unlock;
END_REGION

REGION Network 7: fDoor4 monitoring
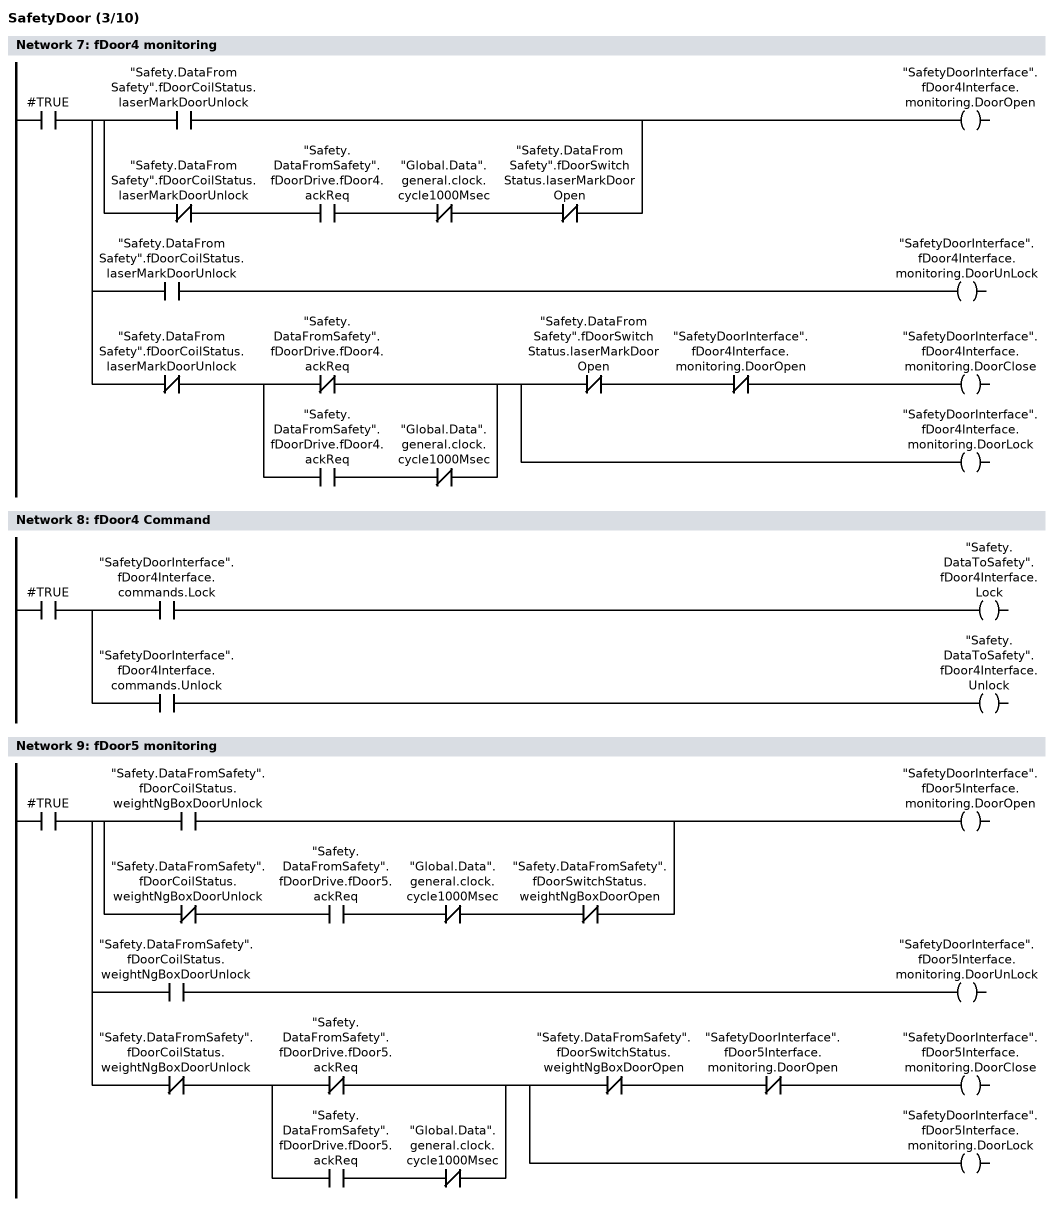
   RUNG wire#powerrail
      Contact( #TRUE )
      wire#w1
      Contact( "Safety.DataFromSafety".fDoorCoilStatus.laserMarkDoorUnlock )
      wire#w2
      Coil( "SafetyDoorInterface".fDoor4Interface.monitoring.DoorOpen )
   END_RUNG
   RUNG wire#w1
      I_Contact( "Safety.DataFromSafety".fDoorCoilStatus.laserMarkDoorUnlock )
      Contact( "Safety.DataFromSafety".fDoorDrive.fDoor4.ackReq )
      I_Contact( "Global.Data".general.clock.cycle1000Msec )
      I_Contact( "Safety.DataFromSafety".fDoorSwitchStatus.laserMarkDoorOpen )
   END_RUNG wire#w2
   RUNG wire#w1
      Contact( "Safety.DataFromSafety".fDoorCoilStatus.laserMarkDoorUnlock )
      Coil( "SafetyDoorInterface".fDoor4Interface.monitoring.DoorUnLock )
   END_RUNG
   RUNG wire#w1
      I_Contact( "Safety.DataFromSafety".fDoorCoilStatus.laserMarkDoorUnlock )
      wire#w3
      I_Contact( "Safety.DataFromSafety".fDoorDrive.fDoor4.ackReq )
      wire#w4
      I_Contact( "Safety.DataFromSafety".fDoorSwitchStatus.laserMarkDoorOpen )
      I_Contact( "SafetyDoorInterface".fDoor4Interface.monitoring.DoorOpen )
      Coil( "SafetyDoorInterface".fDoor4Interface.monitoring.DoorClose )
   END_RUNG
   RUNG wire#w3
      Contact( "Safety.DataFromSafety".fDoorDrive.fDoor4.ackReq )
      I_Contact( "Global.Data".general.clock.cycle1000Msec )
   END_RUNG wire#w4
   RUNG wire#w4
      Coil( "SafetyDoorInterface".fDoor4Interface.monitoring.DoorLock )
   END_RUNG
   // the same network as SCL:
   "SafetyDoorInterface".fDoor4Interface.monitoring.DoorOpen := #TRUE AND ("Safety.DataFromSafety".fDoorCoilStatus.laserMarkDoorUnlock OR (NOT "Safety.DataFromSafety".fDoorCoilStatus.laserMarkDoorUnlock AND "Safety.DataFromSafety".fDoorDrive.fDoor4.ackReq AND NOT "Global.Data".general.clock.cycle1000Msec AND NOT "Safety.DataFromSafety".fDoorSwitchStatus.laserMarkDoorOpen));
   "SafetyDoorInterface".fDoor4Interface.monitoring.DoorUnLock := #TRUE AND "Safety.DataFromSafety".fDoorCoilStatus.laserMarkDoorUnlock;
   #_w1 := #TRUE AND NOT "Safety.DataFromSafety".fDoorCoilStatus.laserMarkDoorUnlock AND (NOT "Safety.DataFromSafety".fDoorDrive.fDoor4.ackReq OR ("Safety.DataFromSafety".fDoorDrive.fDoor4.ackReq AND NOT "Global.Data".general.clock.cycle1000Msec));
   "SafetyDoorInterface".fDoor4Interface.monitoring.DoorClose := #_w1 AND NOT "Safety.DataFromSafety".fDoorSwitchStatus.laserMarkDoorOpen AND NOT "SafetyDoorInterface".fDoor4Interface.monitoring.DoorOpen;
   "SafetyDoorInterface".fDoor4Interface.monitoring.DoorLock := #_w1;
END_REGION

REGION Network 8: fDoor4 Command
   RUNG wire#powerrail
      Contact( #TRUE )
      wire#w1
      Contact( "SafetyDoorInterface".fDoor4Interface.commands.Lock )
      Coil( "Safety.DataToSafety".fDoor4Interface.Lock )
   END_RUNG
   RUNG wire#w1
      Contact( "SafetyDoorInterface".fDoor4Interface.commands.Unlock )
      Coil( "Safety.DataToSafety".fDoor4Interface.Unlock )
   END_RUNG
   // the same network as SCL:
   "Safety.DataToSafety".fDoor4Interface.Lock := #TRUE AND "SafetyDoorInterface".fDoor4Interface.commands.Lock;
   "Safety.DataToSafety".fDoor4Interface.Unlock := #TRUE AND "SafetyDoorInterface".fDoor4Interface.commands.Unlock;
END_REGION

